LIN {X -0.079,Y -462.079,Z 459.993,A 0.000,B 0.000,C 90.000,E1 214.659} C_DIS
LIN {X 0.017,Y -457.566,Z 459.980,A 0.000,B 0.000,C 90.000,E1 212.418} C_DIS
LIN {X -0.236,Y -453.208,Z 459.968,A 0.000,B 0.000,C 90.000,E1 210.207} C_DIS
LIN {X 0.089,Y -449.505,Z 459.957,A 0.000,B 0.000,C 90.000,E1 208.231} C_DIS
LIN {X 0.041,Y -446.412,Z 459.948,A 0.000,B 0.000,C 90.000,E1 206.616} C_DIS
LIN {X 0.179,Y -442.573,Z 459.937,A 0.000,B 0.000,C 90.000,E1 204.643} C_DIS
LIN {X -0.081,Y -440.644,Z 459.932,A 0.000,B 0.000,C 90.000,E1 203.695} C_DIS
LIN {X -0.199,Y -436.151,Z 459.919,A 0.000,B 0.000,C 90.000,E1 201.408} C_DIS
LIN {X -0.233,Y -433.117,Z 459.910,A 0.000,B 0.000,C 90.000,E1 199.758} C_DIS
LIN {X -0.033,Y -429.082,Z 459.897,A 0.000,B 0.000,C 90.000,E1 197.402} C_DIS
LIN {X 0.001,Y -424.902,Z 459.882,A 0.000,B 0.000,C 90.000,E1 194.717} C_DIS
LIN {X -0.050,Y -422.064,Z 459.871,A 0.000,B 0.000,C 90.000,E1 192.703} C_DIS
LIN {X -0.165,Y -418.201,Z 459.854,A 0.000,B 0.000,C 90.000,E1 189.670} C_DIS
LIN {X 0.173,Y -415.396,Z 459.840,A 0.000,B 0.000,C 90.000,E1 187.239} C_DIS
LIN {X -0.106,Y -413.960,Z 459.833,A 0.000,B 0.000,C 90.000,E1 185.910} C_DIS
LIN {X -0.021,Y -411.212,Z 459.818,A 0.000,B 0.000,C 90.000,E1 183.154} C_DIS
LIN {X -0.018,Y -409.551,Z 459.806,A 0.000,B 0.000,C 90.000,E1 181.088} C_DIS
LIN {X -0.128,Y -407.489,Z 459.787,A 0.000,B 0.000,C 90.000,E1 177.650} C_DIS
LIN {X 0.157,Y -406.307,Z 459.766,A 0.000,B 0.000,C 90.000,E1 173.799} C_DIS
LIN {X 0.171,Y -406.510,Z 459.745,A 0.000,B 0.000,C 90.000,E1 169.982} C_DIS
LIN {X 0.162,Y -407.845,Z 459.723,A 0.000,B 0.000,C 90.000,E1 166.172} C_DIS
LIN {X 0.133,Y -408.980,Z 459.712,A 0.000,B 0.000,C 90.000,E1 164.102} C_DIS
LIN {X 0.093,Y -411.915,Z 459.691,A 0.000,B 0.000,C 90.000,E1 160.315} C_DIS
LIN {X -0.064,Y -414.691,Z 459.676,A 0.000,B 0.000,C 90.000,E1 157.592} C_DIS
LIN {X 0.044,Y -417.933,Z 459.660,A 0.000,B 0.000,C 90.000,E1 154.845} C_DIS
LIN {X 0.167,Y -420.127,Z 459.651,A 0.000,B 0.000,C 90.000,E1 153.127} C_DIS
LIN {X -0.114,Y -423.324,Z 459.638,A 0.000,B 0.000,C 90.000,E1 150.795} C_DIS
LIN {X 0.121,Y -426.091,Z 459.626,A 0.000,B 0.000,C 90.000,E1 148.742} C_DIS
LIN {X -0.070,Y -428.532,Z 459.617,A 0.000,B 0.000,C 90.000,E1 147.089} C_DIS
LIN {X 0.148,Y -431.633,Z 459.606,A 0.000,B 0.000,C 90.000,E1 145.055} C_DIS
LIN {X -0.120,Y -435.369,Z 459.593,A 0.000,B 0.000,C 90.000,E1 142.763} C_DIS
LIN {X -0.066,Y -439.785,Z 459.578,A 0.000,B 0.000,C 90.000,E1 140.114} C_DIS
LIN {X -0.206,Y -443.193,Z 459.567,A 0.000,B 0.000,C 90.000,E1 138.162} C_DIS
LIN {X 0.028,Y -445.355,Z 459.560,A 0.000,B 0.000,C 90.000,E1 136.824} C_DIS
LIN {X -0.015,Y -447.307,Z 459.553,A 0.000,B 0.000,C 90.000,E1 135.526} C_DIS
LIN {X -0.039,Y -448.476,Z 459.548,A 0.000,B 0.000,C 90.000,E1 134.555} C_DIS
LIN {X 0.276,Y -449.230,Z 459.544,A 0.000,B 0.000,C 90.000,E1 133.866} C_DIS
LIN {X -0.030,Y -450.411,Z 459.537,A 0.000,B 0.000,C 90.000,E1 132.609} C_DIS
LIN {X 0.014,Y -451.134,Z 459.530,A 0.000,B 0.000,C 90.000,E1 131.310} C_DIS
LIN {X 0.068,Y -451.303,Z 459.524,A 0.000,B 0.000,C 90.000,E1 130.334} C_DIS
LIN {X -0.221,Y -451.124,Z 459.521,A 0.000,B 0.000,C 90.000,E1 129.725} C_DIS
LIN {X 0.119,Y -450.766,Z 459.517,A 0.000,B 0.000,C 90.000,E1 129.036} C_DIS
LIN {X 0.172,Y -450.342,Z 459.513,A 0.000,B 0.000,C 90.000,E1 128.382} C_DIS
LIN {X -0.003,Y -448.898,Z 459.506,A 0.000,B 0.000,C 90.000,E1 127.111} C_DIS
LIN {X 0.008,Y -447.522,Z 459.501,A 0.000,B 0.000,C 90.000,E1 126.137} C_DIS
LIN {X -0.229,Y -446.452,Z 459.497,A 0.000,B 0.000,C 90.000,E1 125.518} C_DIS
LIN {X -0.154,Y -444.523,Z 459.492,A 0.000,B 0.000,C 90.000,E1 124.532} C_DIS
LIN {X -0.057,Y -441.550,Z 459.485,A 0.000,B 0.000,C 90.000,E1 123.214} C_DIS
LIN {X 0.124,Y -438.283,Z 459.477,A 0.000,B 0.000,C 90.000,E1 121.878} C_DIS
LIN {X -0.117,Y -434.841,Z 459.470,A 0.000,B 0.000,C 90.000,E1 120.590} C_DIS
LIN {X 0.122,Y -432.255,Z 459.465,A 0.000,B 0.000,C 90.000,E1 119.617} C_DIS
LIN {X 0.083,Y -432.255,Z 459.465,A 0.000,B 0.000,C 90.000,E1 119.617} C_DIS
LIN {X 0.136,Y -441.772,Z 459.444,A 0.000,B 0.000,C 90.000,E1 115.924} C_DIS
LIN {X 0.059,Y -444.699,Z 459.439,A 0.000,B 0.000,C 90.000,E1 114.951} C_DIS
LIN {X 0.031,Y -454.671,Z 459.415,A 0.000,B 0.000,C 90.000,E1 110.737} C_DIS
LIN {X 0.153,Y -457.324,Z 459.410,A 0.000,B 0.000,C 90.000,E1 109.758} C_DIS
LIN {X -0.209,Y -465.949,Z 459.387,A 0.000,B 0.000,C 90.000,E1 105.662} C_DIS
LIN {X -0.038,Y -467.513,Z 459.383,A 0.000,B 0.000,C 90.000,E1 105.009} C_DIS
LIN {X -0.234,Y -468.096,Z 459.382,A 0.000,B 0.000,C 90.000,E1 104.717} C_DIS
LIN {X -0.094,Y -475.756,Z 459.357,A 0.000,B 0.000,C 90.000,E1 100.310} C_DIS
LIN {X 0.211,Y -476.285,Z 459.356,A 0.000,B 0.000,C 90.000,E1 99.962} C_DIS
LIN {X 0.208,Y -479.372,Z 459.340,A 0.000,B 0.000,C 90.000,E1 97.239} C_DIS
LIN {X 0.188,Y -558.722,Z 459.340,A 0.000,B 0.000,C 90.000,E1 97.239} C_DIS
LIN {X 0.091,Y -564.116,Z 459.340,A 0.000,B 0.000,C 90.000,E1 97.182} C_DIS
LIN {X 0.113,Y -570.120,Z 459.339,A 0.000,B 0.000,C 90.000,E1 97.068} C_DIS
LIN {X -0.229,Y -576.419,Z 459.339,A 0.000,B 0.000,C 90.000,E1 96.947} C_DIS
LIN {X 0.097,Y -582.845,Z 459.337,A 0.000,B 0.000,C 90.000,E1 96.720} C_DIS
LIN {X 0.040,Y -589.213,Z 459.336,A 0.000,B 0.000,C 90.000,E1 96.486} C_DIS
LIN {X 0.176,Y -595.796,Z 459.335,A 0.000,B 0.000,C 90.000,E1 96.201} C_DIS
LIN {X -0.029,Y -601.591,Z 459.333,A 0.000,B 0.000,C 90.000,E1 95.910} C_DIS
LIN {X -0.209,Y -607.593,Z 459.331,A 0.000,B 0.000,C 90.000,E1 95.568} C_DIS
LIN {X -0.076,Y -613.091,Z 459.329,A 0.000,B 0.000,C 90.000,E1 95.163} C_DIS
LIN {X 0.014,Y -614.544,Z 459.328,A 0.000,B 0.000,C 90.000,E1 95.049} C_DIS
LIN {X -0.034,Y -620.912,Z 459.325,A 0.000,B 0.000,C 90.000,E1 94.473} C_DIS
LIN {X 0.204,Y -625.161,Z 459.322,A 0.000,B 0.000,C 90.000,E1 93.955} C_DIS
LIN {X -0.090,Y -627.282,Z 459.321,A 0.000,B 0.000,C 90.000,E1 93.726} C_DIS
LIN {X 0.250,Y -628.777,Z 459.319,A 0.000,B 0.000,C 90.000,E1 93.440} C_DIS
LIN {X -0.269,Y -631.451,Z 459.316,A 0.000,B 0.000,C 90.000,E1 92.980} C_DIS
LIN {X -0.179,Y -633.775,Z 459.314,A 0.000,B 0.000,C 90.000,E1 92.465} C_DIS
LIN {X -0.306,Y -635.760,Z 459.309,A 0.000,B 0.000,C 90.000,E1 91.718} C_DIS
LIN {X -0.181,Y -636.632,Z 459.307,A 0.000,B 0.000,C 90.000,E1 91.203} C_DIS
LIN {X -0.048,Y -637.073,Z 459.304,A 0.000,B 0.000,C 90.000,E1 90.688} C_DIS
LIN {X 0.091,Y -637.071,Z 459.301,A 0.000,B 0.000,C 90.000,E1 90.172} C_DIS
LIN {X -0.158,Y -636.918,Z 459.300,A 0.000,B 0.000,C 90.000,E1 89.943} C_DIS
LIN {X -0.019,Y -636.261,Z 459.297,A 0.000,B 0.000,C 90.000,E1 89.427} C_DIS
LIN {X 0.114,Y -635.024,Z 459.294,A 0.000,B 0.000,C 90.000,E1 88.912} C_DIS
LIN {X 0.238,Y -633.501,Z 459.291,A 0.000,B 0.000,C 90.000,E1 88.396} C_DIS
LIN {X -0.001,Y -632.517,Z 459.290,A 0.000,B 0.000,C 90.000,E1 88.165} C_DIS
LIN {X 0.107,Y -629.929,Z 459.287,A 0.000,B 0.000,C 90.000,E1 87.650} C_DIS
LIN {X 0.050,Y -626.107,Z 459.284,A 0.000,B 0.000,C 90.000,E1 87.020} C_DIS
LIN {X -0.153,Y -620.658,Z 459.279,A 0.000,B 0.000,C 90.000,E1 86.274} C_DIS
LIN {X -0.250,Y -615.157,Z 459.276,A 0.000,B 0.000,C 90.000,E1 85.641} C_DIS
LIN {X -0.065,Y -609.946,Z 459.273,A 0.000,B 0.000,C 90.000,E1 85.122} C_DIS
LIN {X -0.133,Y -608.649,Z 459.272,A 0.000,B 0.000,C 90.000,E1 85.008} C_DIS
LIN {X -0.109,Y -603.026,Z 459.270,A 0.000,B 0.000,C 90.000,E1 84.546} C_DIS
LIN {X 0.081,Y -598.091,Z 459.268,A 0.000,B 0.000,C 90.000,E1 84.204} C_DIS
LIN {X -0.141,Y -594.766,Z 459.267,A 0.000,B 0.000,C 90.000,E1 84.033} C_DIS
LIN {X -0.035,Y -588.527,Z 459.265,A 0.000,B 0.000,C 90.000,E1 83.685} C_DIS
LIN {X -0.071,Y -585.000,Z 459.264,A 0.000,B 0.000,C 90.000,E1 83.514} C_DIS
LIN {X -0.245,Y -583.090,Z 459.264,A 0.000,B 0.000,C 90.000,E1 83.451} C_DIS
LIN {X 0.093,Y -577.795,Z 459.262,A 0.000,B 0.000,C 90.000,E1 83.223} C_DIS
LIN {X -0.016,Y -571.567,Z 459.261,A 0.000,B 0.000,C 90.000,E1 83.053} C_DIS
LIN {X 0.061,Y -564.953,Z 459.261,A 0.000,B 0.000,C 90.000,E1 82.932} C_DIS
LIN {X 0.160,Y -559.170,Z 459.261,A 0.000,B 0.000,C 90.000,E1 82.875} C_DIS
LIN {X 0.104,Y -484.840,Z 459.261,A 0.000,B 0.000,C 90.000,E1 82.875} C_DIS
LIN {X -0.113,Y -484.690,Z 459.254,A 0.000,B 0.000,C 90.000,E1 81.659} C_DIS
LIN {X -0.099,Y -483.703,Z 459.249,A 0.000,B 0.000,C 90.000,E1 80.735} C_DIS
LIN {X 0.265,Y -480.630,Z 459.228,A 0.000,B 0.000,C 90.000,E1 76.992} C_DIS
LIN {X 0.123,Y -480.315,Z 459.226,A 0.000,B 0.000,C 90.000,E1 76.700} C_DIS
LIN {X 0.026,Y -474.131,Z 459.200,A 0.000,B 0.000,C 90.000,E1 72.054} C_DIS
LIN {X -0.105,Y -465.601,Z 459.172,A 0.000,B 0.000,C 90.000,E1 67.050} C_DIS
LIN {X -0.108,Y -458.658,Z 459.154,A 0.000,B 0.000,C 90.000,E1 63.768} C_DIS
LIN {X -0.147,Y -458.658,Z 459.154,A 0.000,B 0.000,C 90.000,E1 63.768} C_DIS
LIN {X -0.198,Y -466.432,Z 459.148,A 0.000,B 0.000,C 90.000,E1 62.615} C_DIS
LIN {X -0.201,Y -473.768,Z 459.142,A 0.000,B 0.000,C 90.000,E1 61.513} C_DIS
LIN {X 0.126,Y -480.526,Z 459.136,A 0.000,B 0.000,C 90.000,E1 60.383} C_DIS
LIN {X 0.085,Y -484.924,Z 459.131,A 0.000,B 0.000,C 90.000,E1 59.616} C_DIS
LIN {X 0.123,Y -488.077,Z 459.128,A 0.000,B 0.000,C 90.000,E1 58.997} C_DIS
LIN {X -0.021,Y -491.497,Z 459.124,A 0.000,B 0.000,C 90.000,E1 58.250} C_DIS
LIN {X -0.189,Y -493.935,Z 459.120,A 0.000,B 0.000,C 90.000,E1 57.661} C_DIS
LIN {X -0.077,Y -495.986,Z 459.117,A 0.000,B 0.000,C 90.000,E1 57.041} C_DIS
LIN {X -0.087,Y -498.471,Z 459.112,A 0.000,B 0.000,C 90.000,E1 56.135} C_DIS
LIN {X 0.063,Y -499.755,Z 459.109,A 0.000,B 0.000,C 90.000,E1 55.515} C_DIS
LIN {X 0.098,Y -501.142,Z 459.103,A 0.000,B 0.000,C 90.000,E1 54.609} C_DIS
LIN {X 0.147,Y -502.283,Z 459.098,A 0.000,B 0.000,C 90.000,E1 53.703} C_DIS
LIN {X -0.200,Y -502.907,Z 459.094,A 0.000,B 0.000,C 90.000,E1 52.844} C_DIS
LIN {X 0.053,Y -503.314,Z 459.087,A 0.000,B 0.000,C 90.000,E1 51.618} C_DIS
LIN {X 0.029,Y -503.403,Z 459.082,A 0.000,B 0.000,C 90.000,E1 50.723} C_DIS
LIN {X 0.124,Y -503.387,Z 459.079,A 0.000,B 0.000,C 90.000,E1 50.114} C_DIS
LIN {X 0.104,Y -503.125,Z 459.074,A 0.000,B 0.000,C 90.000,E1 49.218} C_DIS
LIN {X -0.331,Y -502.312,Z 459.064,A 0.000,B 0.000,C 90.000,E1 47.472} C_DIS
LIN {X 0.177,Y -501.600,Z 459.057,A 0.000,B 0.000,C 90.000,E1 46.215} C_DIS
LIN {X -0.185,Y -500.627,Z 459.049,A 0.000,B 0.000,C 90.000,E1 44.757} C_DIS
LIN {X -0.065,Y -499.708,Z 459.042,A 0.000,B 0.000,C 90.000,E1 43.542} C_DIS
LIN {X -0.108,Y -498.547,Z 459.034,A 0.000,B 0.000,C 90.000,E1 42.043} C_DIS
LIN {X 0.050,Y -497.041,Z 459.023,A 0.000,B 0.000,C 90.000,E1 40.216} C_DIS
LIN {X 0.236,Y -495.466,Z 459.013,A 0.000,B 0.000,C 90.000,E1 38.382} C_DIS
LIN {X 0.086,Y -493.825,Z 459.003,A 0.000,B 0.000,C 90.000,E1 36.583} C_DIS
LIN {X -0.094,Y -492.591,Z 458.997,A 0.000,B 0.000,C 90.000,E1 35.391} C_DIS
LIN {X -0.038,Y -490.933,Z 458.988,A 0.000,B 0.000,C 90.000,E1 33.865} C_DIS
LIN {X -0.018,Y -489.233,Z 458.980,A 0.000,B 0.000,C 90.000,E1 32.339} C_DIS
LIN {X 0.114,Y -487.317,Z 458.971,A 0.000,B 0.000,C 90.000,E1 30.797} C_DIS
LIN {X -0.028,Y -485.783,Z 458.964,A 0.000,B 0.000,C 90.000,E1 29.589} C_DIS
LIN {X -0.221,Y -483.471,Z 458.954,A 0.000,B 0.000,C 90.000,E1 27.769} C_DIS
LIN {X -0.054,Y -480.630,Z 458.940,A 0.000,B 0.000,C 90.000,E1 25.283} C_DIS
LIN {X -0.176,Y -478.269,Z 458.927,A 0.000,B 0.000,C 90.000,E1 22.823} C_DIS
LIN {X 0.159,Y -476.710,Z 458.915,A 0.000,B 0.000,C 90.000,E1 20.610} C_DIS
LIN {X -0.137,Y -475.497,Z 458.904,A 0.000,B 0.000,C 90.000,E1 18.779} C_DIS
LIN {X -0.130,Y -474.555,Z 458.896,A 0.000,B 0.000,C 90.000,E1 17.221} C_DIS
LIN {X 0.096,Y -473.109,Z 458.883,A 0.000,B 0.000,C 90.000,E1 15.009} C_DIS
LIN {X -0.097,Y -471.382,Z 458.864,A 0.000,B 0.000,C 90.000,E1 11.591} C_DIS
LIN {X 0.198,Y -470.425,Z 458.845,A 0.000,B 0.000,C 90.000,E1 8.106} C_DIS
LIN {X -0.196,Y -470.501,Z 458.826,A 0.000,B 0.000,C 90.000,E1 4.702} C_DIS
LIN {X -0.231,Y -472.150,Z 458.803,A 0.000,B 0.000,C 90.000,E1 0.630} C_DIS
LIN {X 0.218,Y -473.164,Z 458.795,A 0.000,B 0.000,C 90.000,E1 359.141} C_DIS
LIN {X 0.223,Y -475.718,Z 458.780,A 0.000,B 0.000,C 90.000,E1 356.331} C_DIS
LIN {X -0.096,Y -479.014,Z 458.764,A 0.000,B 0.000,C 90.000,E1 353.571} C_DIS
LIN {X 0.150,Y -481.944,Z 458.752,A 0.000,B 0.000,C 90.000,E1 351.376} C_DIS
LIN {X 0.158,Y -485.257,Z 458.740,A 0.000,B 0.000,C 90.000,E1 349.218} C_DIS
LIN {X -0.088,Y -491.443,Z 458.722,A 0.000,B 0.000,C 90.000,E1 345.880} C_DIS
LIN {X 0.038,Y -496.067,Z 458.710,A 0.000,B 0.000,C 90.000,E1 343.740} C_DIS
LIN {X -0.044,Y -501.143,Z 458.698,A 0.000,B 0.000,C 90.000,E1 341.638} C_DIS
LIN {X 0.165,Y -506.451,Z 458.686,A 0.000,B 0.000,C 90.000,E1 339.518} C_DIS
LIN {X 0.096,Y -511.096,Z 458.676,A 0.000,B 0.000,C 90.000,E1 337.741} C_DIS
LIN {X 0.053,Y -515.667,Z 458.667,A 0.000,B 0.000,C 90.000,E1 335.973} C_DIS
LIN {X -0.235,Y -519.412,Z 458.658,A 0.000,B 0.000,C 90.000,E1 334.537} C_DIS
LIN {X 0.140,Y -523.946,Z 458.649,A 0.000,B 0.000,C 90.000,E1 332.743} C_DIS
LIN {X -0.209,Y -529.892,Z 458.636,A 0.000,B 0.000,C 90.000,E1 330.461} C_DIS
LIN {X 0.159,Y -535.227,Z 458.625,A 0.000,B 0.000,C 90.000,E1 328.408} C_DIS
LIN {X 0.023,Y -539.779,Z 458.615,A 0.000,B 0.000,C 90.000,E1 326.707} C_DIS
LIN {X -0.188,Y -543.602,Z 458.607,A 0.000,B 0.000,C 90.000,E1 325.308} C_DIS
LIN {X -0.240,Y -549.057,Z 458.596,A 0.000,B 0.000,C 90.000,E1 323.336} C_DIS
LIN {X 0.102,Y -553.814,Z 458.587,A 0.000,B 0.000,C 90.000,E1 321.618} C_DIS
LIN {X 0.196,Y -560.142,Z 458.574,A 0.000,B 0.000,C 90.000,E1 319.380} C_DIS
LIN {X -0.157,Y -564.970,Z 458.565,A 0.000,B 0.000,C 90.000,E1 317.757} C_DIS
LIN {X -0.106,Y -568.885,Z 458.558,A 0.000,B 0.000,C 90.000,E1 316.377} C_DIS
LIN {X 0.215,Y -574.285,Z 458.547,A 0.000,B 0.000,C 90.000,E1 314.433} C_DIS
LIN {X -0.267,Y -578.948,Z 458.538,A 0.000,B 0.000,C 90.000,E1 312.852} C_DIS
LIN {X 0.039,Y -582.833,Z 458.530,A 0.000,B 0.000,C 90.000,E1 311.472} C_DIS
LIN {X -0.033,Y -586.689,Z 458.523,A 0.000,B 0.000,C 90.000,E1 310.135} C_DIS
LIN {X -0.095,Y -589.734,Z 458.517,A 0.000,B 0.000,C 90.000,E1 309.072} C_DIS
LIN {X 0.016,Y -593.385,Z 458.510,A 0.000,B 0.000,C 90.000,E1 307.729} C_DIS
LIN {X 0.066,Y -596.294,Z 458.504,A 0.000,B 0.000,C 90.000,E1 306.664} C_DIS
LIN {X -0.092,Y -599.857,Z 458.496,A 0.000,B 0.000,C 90.000,E1 305.358} C_DIS
LIN {X 0.194,Y -602.579,Z 458.491,A 0.000,B 0.000,C 90.000,E1 304.278} C_DIS
LIN {X 0.031,Y -605.197,Z 458.485,A 0.000,B 0.000,C 90.000,E1 303.245} C_DIS
LIN {X -0.100,Y -607.702,Z 458.479,A 0.000,B 0.000,C 90.000,E1 302.212} C_DIS
LIN {X -0.307,Y -611.284,Z 458.470,A 0.000,B 0.000,C 90.000,E1 300.669} C_DIS
LIN {X 0.114,Y -614.013,Z 458.463,A 0.000,B 0.000,C 90.000,E1 299.333} C_DIS
LIN {X 0.277,Y -616.687,Z 458.456,A 0.000,B 0.000,C 90.000,E1 298.025} C_DIS
LIN {X 0.189,Y -619.833,Z 458.447,A 0.000,B 0.000,C 90.000,E1 296.488} C_DIS
LIN {X 0.171,Y -621.298,Z 458.443,A 0.000,B 0.000,C 90.000,E1 295.720} C_DIS
LIN {X -0.093,Y -623.968,Z 458.434,A 0.000,B 0.000,C 90.000,E1 294.207} C_DIS
LIN {X 0.258,Y -625.952,Z 458.427,A 0.000,B 0.000,C 90.000,E1 292.898} C_DIS
LIN {X -0.166,Y -628.104,Z 458.419,A 0.000,B 0.000,C 90.000,E1 291.408} C_DIS
LIN {X 0.018,Y -629.794,Z 458.412,A 0.000,B 0.000,C 90.000,E1 290.120} C_DIS
LIN {X 0.019,Y -631.360,Z 458.405,A 0.000,B 0.000,C 90.000,E1 288.852} C_DIS
LIN {X 0.050,Y -632.768,Z 458.398,A 0.000,B 0.000,C 90.000,E1 287.583} C_DIS
LIN {X -0.088,Y -634.202,Z 458.389,A 0.000,B 0.000,C 90.000,E1 286.079} C_DIS
LIN {X -0.017,Y -634.817,Z 458.385,A 0.000,B 0.000,C 90.000,E1 285.315} C_DIS
LIN {X -0.297,Y -635.887,Z 458.377,A 0.000,B 0.000,C 90.000,E1 283.828} C_DIS
LIN {X 0.074,Y -636.469,Z 458.370,A 0.000,B 0.000,C 90.000,E1 282.535} C_DIS
LIN {X 0.002,Y -636.857,Z 458.364,A 0.000,B 0.000,C 90.000,E1 281.535} C_DIS
LIN {X 0.257,Y -637.126,Z 458.357,A 0.000,B 0.000,C 90.000,E1 280.254} C_DIS
LIN {X -0.112,Y -637.081,Z 458.350,A 0.000,B 0.000,C 90.000,E1 279.029} C_DIS
LIN {X 0.229,Y -636.921,Z 458.345,A 0.000,B 0.000,C 90.000,E1 277.992} C_DIS
LIN {X 0.023,Y -636.491,Z 458.339,A 0.000,B 0.000,C 90.000,E1 277.004} C_DIS
LIN {X -0.074,Y -636.007,Z 458.335,A 0.000,B 0.000,C 90.000,E1 276.258} C_DIS
LIN {X 0.258,Y -635.175,Z 458.329,A 0.000,B 0.000,C 90.000,E1 275.220} C_DIS
LIN {X 0.153,Y -634.309,Z 458.325,A 0.000,B 0.000,C 90.000,E1 274.473} C_DIS
LIN {X -0.223,Y -632.945,Z 458.319,A 0.000,B 0.000,C 90.000,E1 273.498} C_DIS
LIN {X -0.250,Y -630.965,Z 458.312,A 0.000,B 0.000,C 90.000,E1 272.236} C_DIS
LIN {X 0.314,Y -628.647,Z 458.305,A 0.000,B 0.000,C 90.000,E1 270.917} C_DIS
LIN {X 0.194,Y -626.139,Z 458.298,A 0.000,B 0.000,C 90.000,E1 269.656} C_DIS
LIN {X 0.030,Y -623.442,Z 458.291,A 0.000,B 0.000,C 90.000,E1 268.396} C_DIS
LIN {X -0.165,Y -620.490,Z 458.284,A 0.000,B 0.000,C 90.000,E1 267.135} C_DIS
LIN {X 0.249,Y -617.421,Z 458.277,A 0.000,B 0.000,C 90.000,E1 265.812} C_DIS
LIN {X -0.026,Y -615.558,Z 458.273,A 0.000,B 0.000,C 90.000,E1 265.065} C_DIS
LIN {X 0.307,Y -612.250,Z 458.265,A 0.000,B 0.000,C 90.000,E1 263.742} C_DIS
LIN {X -0.295,Y -609.623,Z 458.260,A 0.000,B 0.000,C 90.000,E1 262.761} C_DIS
LIN {X -0.001,Y -606.148,Z 458.252,A 0.000,B 0.000,C 90.000,E1 261.432} C_DIS
LIN {X -0.275,Y -602.664,Z 458.245,A 0.000,B 0.000,C 90.000,E1 260.151} C_DIS
LIN {X 0.273,Y -599.738,Z 458.239,A 0.000,B 0.000,C 90.000,E1 259.050} C_DIS
LIN {X 0.006,Y -594.420,Z 458.229,A 0.000,B 0.000,C 90.000,E1 257.229} C_DIS
LIN {X 0.233,Y -590.449,Z 458.222,A 0.000,B 0.000,C 90.000,E1 255.880} C_DIS
LIN {X 0.276,Y -587.280,Z 458.216,A 0.000,B 0.000,C 90.000,E1 254.810} C_DIS
LIN {X 0.278,Y -584.000,Z 458.210,A 0.000,B 0.000,C 90.000,E1 253.740} C_DIS
LIN {X 0.228,Y -580.693,Z 458.204,A 0.000,B 0.000,C 90.000,E1 252.670} C_DIS
LIN {X -0.244,Y -577.325,Z 458.198,A 0.000,B 0.000,C 90.000,E1 251.638} C_DIS
LIN {X -0.210,Y -573.874,Z 458.192,A 0.000,B 0.000,C 90.000,E1 250.550} C_DIS
LIN {X -0.031,Y -570.334,Z 458.186,A 0.000,B 0.000,C 90.000,E1 249.444} C_DIS
LIN {X -0.295,Y -565.802,Z 458.178,A 0.000,B 0.000,C 90.000,E1 248.103} C_DIS
LIN {X -0.016,Y -561.956,Z 458.172,A 0.000,B 0.000,C 90.000,E1 246.975} C_DIS
LIN {X -0.225,Y -556.948,Z 458.164,A 0.000,B 0.000,C 90.000,E1 245.613} C_DIS
LIN {X 0.159,Y -552.860,Z 458.158,A 0.000,B 0.000,C 90.000,E1 244.460} C_DIS
LIN {X 0.006,Y -547.692,Z 458.150,A 0.000,B 0.000,C 90.000,E1 243.076} C_DIS
LIN {X -0.004,Y -540.403,Z 458.139,A 0.000,B 0.000,C 90.000,E1 241.101} C_DIS
LIN {X 0.117,Y -535.302,Z 458.132,A 0.000,B 0.000,C 90.000,E1 239.665} C_DIS
LIN {X 0.100,Y -529.219,Z 458.122,A 0.000,B 0.000,C 90.000,E1 237.946} C_DIS
LIN {X 0.065,Y -523.158,Z 458.112,A 0.000,B 0.000,C 90.000,E1 236.215} C_DIS
LIN {X -0.037,Y -518.073,Z 458.104,A 0.000,B 0.000,C 90.000,E1 234.769} C_DIS
LIN {X -0.015,Y -511.827,Z 458.095,A 0.000,B 0.000,C 90.000,E1 233.004} C_DIS
LIN {X -0.243,Y -500.491,Z 458.075,A 0.000,B 0.000,C 90.000,E1 229.461} C_DIS
LIN {X -0.057,Y -495.153,Z 458.065,A 0.000,B 0.000,C 90.000,E1 227.634} C_DIS
LIN {X 0.145,Y -489.132,Z 458.053,A 0.000,B 0.000,C 90.000,E1 225.486} C_DIS
LIN {X -0.159,Y -483.326,Z 458.041,A 0.000,B 0.000,C 90.000,E1 223.380} C_DIS
LIN {X -0.037,Y -478.500,Z 458.031,A 0.000,B 0.000,C 90.000,E1 221.515} C_DIS
LIN {X -0.106,Y -472.498,Z 458.017,A 0.000,B 0.000,C 90.000,E1 219.036} C_DIS
LIN {X 0.081,Y -466.776,Z 458.003,A 0.000,B 0.000,C 90.000,E1 216.503} C_DIS
LIN {X -0.088,Y -463.431,Z 457.994,A 0.000,B 0.000,C 90.000,E1 214.945} C_DIS
LIN {X -0.218,Y -458.209,Z 457.980,A 0.000,B 0.000,C 90.000,E1 212.418} C_DIS
LIN {X 0.167,Y -453.831,Z 457.968,A 0.000,B 0.000,C 90.000,E1 210.129} C_DIS
LIN {X -0.112,Y -450.078,Z 457.957,A 0.000,B 0.000,C 90.000,E1 208.231} C_DIS
LIN {X -0.147,Y -446.989,Z 457.948,A 0.000,B 0.000,C 90.000,E1 206.616} C_DIS
LIN {X -0.136,Y -442.490,Z 457.935,A 0.000,B 0.000,C 90.000,E1 204.335} C_DIS
LIN {X -0.030,Y -437.922,Z 457.922,A 0.000,B 0.000,C 90.000,E1 202.025} C_DIS
LIN {X -0.201,Y -434.232,Z 457.911,A 0.000,B 0.000,C 90.000,E1 200.066} C_DIS
LIN {X 0.165,Y -430.094,Z 457.898,A 0.000,B 0.000,C 90.000,E1 197.692} C_DIS
LIN {X 0.219,Y -425.850,Z 457.884,A 0.000,B 0.000,C 90.000,E1 195.009} C_DIS
LIN {X 0.091,Y -422.938,Z 457.872,A 0.000,B 0.000,C 90.000,E1 193.008} C_DIS
LIN {X 0.097,Y -418.963,Z 457.855,A 0.000,B 0.000,C 90.000,E1 189.962} C_DIS
LIN {X -0.008,Y -416.504,Z 457.844,A 0.000,B 0.000,C 90.000,E1 187.936} C_DIS
LIN {X -0.174,Y -414.304,Z 457.833,A 0.000,B 0.000,C 90.000,E1 185.910} C_DIS
LIN {X -0.077,Y -411.557,Z 457.818,A 0.000,B 0.000,C 90.000,E1 183.154} C_DIS
LIN {X -0.066,Y -409.863,Z 457.806,A 0.000,B 0.000,C 90.000,E1 181.088} C_DIS
LIN {X -0.163,Y -407.814,Z 457.787,A 0.000,B 0.000,C 90.000,E1 177.650} C_DIS
LIN {X 0.101,Y -406.617,Z 457.764,A 0.000,B 0.000,C 90.000,E1 173.457} C_DIS
LIN {X 0.167,Y -406.864,Z 457.745,A 0.000,B 0.000,C 90.000,E1 169.982} C_DIS
LIN {X 0.174,Y -408.233,Z 457.723,A 0.000,B 0.000,C 90.000,E1 166.172} C_DIS
LIN {X 0.155,Y -409.379,Z 457.712,A 0.000,B 0.000,C 90.000,E1 164.102} C_DIS
LIN {X 0.133,Y -412.347,Z 457.691,A 0.000,B 0.000,C 90.000,E1 160.315} C_DIS
LIN {X 0.078,Y -414.761,Z 457.677,A 0.000,B 0.000,C 90.000,E1 157.922} C_DIS
LIN {X 0.032,Y -417.575,Z 457.664,A 0.000,B 0.000,C 90.000,E1 155.537} C_DIS
LIN {X -0.128,Y -420.664,Z 457.651,A 0.000,B 0.000,C 90.000,E1 153.179} C_DIS
LIN {X -0.041,Y -424.416,Z 457.636,A 0.000,B 0.000,C 90.000,E1 150.461} C_DIS
LIN {X -0.153,Y -427.750,Z 457.623,A 0.000,B 0.000,C 90.000,E1 148.122} C_DIS
LIN {X 0.047,Y -431.338,Z 457.610,A 0.000,B 0.000,C 90.000,E1 145.754} C_DIS
LIN {X 0.198,Y -433.507,Z 457.602,A 0.000,B 0.000,C 90.000,E1 144.402} C_DIS
LIN {X 0.059,Y -436.825,Z 457.591,A 0.000,B 0.000,C 90.000,E1 142.431} C_DIS
LIN {X 0.181,Y -440.195,Z 457.580,A 0.000,B 0.000,C 90.000,E1 140.436} C_DIS
LIN {X 0.106,Y -441.952,Z 457.575,A 0.000,B 0.000,C 90.000,E1 139.461} C_DIS
LIN {X -0.002,Y -444.871,Z 457.566,A 0.000,B 0.000,C 90.000,E1 137.838} C_DIS
LIN {X -0.030,Y -446.601,Z 457.560,A 0.000,B 0.000,C 90.000,E1 136.863} C_DIS
LIN {X -0.067,Y -448.602,Z 457.553,A 0.000,B 0.000,C 90.000,E1 135.567} C_DIS
LIN {X -0.071,Y -449.479,Z 457.550,A 0.000,B 0.000,C 90.000,E1 134.919} C_DIS
LIN {X -0.064,Y -450.668,Z 457.544,A 0.000,B 0.000,C 90.000,E1 133.947} C_DIS
LIN {X 0.288,Y -451.958,Z 457.537,A 0.000,B 0.000,C 90.000,E1 132.609} C_DIS
LIN {X 0.019,Y -452.794,Z 457.530,A 0.000,B 0.000,C 90.000,E1 131.353} C_DIS
LIN {X 0.086,Y -452.998,Z 457.524,A 0.000,B 0.000,C 90.000,E1 130.378} C_DIS
LIN {X -0.130,Y -452.771,Z 457.519,A 0.000,B 0.000,C 90.000,E1 129.439} C_DIS
LIN {X 0.225,Y -452.366,Z 457.515,A 0.000,B 0.000,C 90.000,E1 128.749} C_DIS
LIN {X 0.291,Y -451.846,Z 457.512,A 0.000,B 0.000,C 90.000,E1 128.096} C_DIS
LIN {X 0.067,Y -450.752,Z 457.507,A 0.000,B 0.000,C 90.000,E1 127.156} C_DIS
LIN {X -0.170,Y -449.390,Z 457.501,A 0.000,B 0.000,C 90.000,E1 126.217} C_DIS
LIN {X 0.235,Y -448.380,Z 457.498,A 0.000,B 0.000,C 90.000,E1 125.518} C_DIS
LIN {X 0.076,Y -446.440,Z 457.492,A 0.000,B 0.000,C 90.000,E1 124.565} C_DIS
LIN {X 0.089,Y -445.031,Z 457.489,A 0.000,B 0.000,C 90.000,E1 123.913} C_DIS
LIN {X -0.047,Y -441.826,Z 457.481,A 0.000,B 0.000,C 90.000,E1 122.625} C_DIS
LIN {X -0.229,Y -438.395,Z 457.474,A 0.000,B 0.000,C 90.000,E1 121.337} C_DIS
LIN {X -0.093,Y -434.835,Z 457.467,A 0.000,B 0.000,C 90.000,E1 120.001} C_DIS
LIN {X 0.030,Y -432.938,Z 457.463,A 0.000,B 0.000,C 90.000,E1 119.333} C_DIS
LIN {X -0.009,Y -432.938,Z 457.463,A 0.000,B 0.000,C 90.000,E1 119.333} C_DIS
LIN {X -0.098,Y -441.932,Z 457.444,A 0.000,B 0.000,C 90.000,E1 115.899} C_DIS
LIN {X 0.034,Y -444.846,Z 457.438,A 0.000,B 0.000,C 90.000,E1 114.899} C_DIS
LIN {X -0.130,Y -453.953,Z 457.417,A 0.000,B 0.000,C 90.000,E1 111.025} C_DIS
LIN {X 0.152,Y -457.428,Z 457.410,A 0.000,B 0.000,C 90.000,E1 109.704} C_DIS
LIN {X -0.194,Y -466.078,Z 457.387,A 0.000,B 0.000,C 90.000,E1 105.607} C_DIS
LIN {X -0.021,Y -467.647,Z 457.383,A 0.000,B 0.000,C 90.000,E1 104.954} C_DIS
LIN {X 0.174,Y -470.066,Z 457.374,A 0.000,B 0.000,C 90.000,E1 103.355} C_DIS
LIN {X -0.063,Y -475.867,Z 457.357,A 0.000,B 0.000,C 90.000,E1 100.254} C_DIS
LIN {X -0.225,Y -476.334,Z 457.355,A 0.000,B 0.000,C 90.000,E1 99.962} C_DIS
LIN {X -0.113,Y -480.144,Z 457.337,A 0.000,B 0.000,C 90.000,E1 96.720} C_DIS
LIN {X -0.178,Y -559.233,Z 457.337,A 0.000,B 0.000,C 90.000,E1 96.720} C_DIS
LIN {X 0.256,Y -563.077,Z 457.337,A 0.000,B 0.000,C 90.000,E1 96.663} C_DIS
LIN {X 0.255,Y -570.611,Z 457.337,A 0.000,B 0.000,C 90.000,E1 96.549} C_DIS
LIN {X 0.217,Y -577.047,Z 457.336,A 0.000,B 0.000,C 90.000,E1 96.429} C_DIS
LIN {X 0.189,Y -582.818,Z 457.335,A 0.000,B 0.000,C 90.000,E1 96.258} C_DIS
LIN {X 0.128,Y -588.948,Z 457.334,A 0.000,B 0.000,C 90.000,E1 96.030} C_DIS
LIN {X 0.241,Y -595.503,Z 457.332,A 0.000,B 0.000,C 90.000,E1 95.739} C_DIS
LIN {X 0.023,Y -601.509,Z 457.330,A 0.000,B 0.000,C 90.000,E1 95.454} C_DIS
LIN {X -0.064,Y -607.312,Z 457.328,A 0.000,B 0.000,C 90.000,E1 95.106} C_DIS
LIN {X -0.193,Y -611.507,Z 457.327,A 0.000,B 0.000,C 90.000,E1 94.821} C_DIS
LIN {X 0.038,Y -614.311,Z 457.326,A 0.000,B 0.000,C 90.000,E1 94.588} C_DIS
LIN {X -0.068,Y -620.665,Z 457.322,A 0.000,B 0.000,C 90.000,E1 94.012} C_DIS
LIN {X 0.201,Y -623.734,Z 457.320,A 0.000,B 0.000,C 90.000,E1 93.612} C_DIS
LIN {X -0.242,Y -626.536,Z 457.318,A 0.000,B 0.000,C 90.000,E1 93.269} C_DIS
LIN {X 0.276,Y -627.340,Z 457.317,A 0.000,B 0.000,C 90.000,E1 93.094} C_DIS
LIN {X -0.150,Y -629.086,Z 457.315,A 0.000,B 0.000,C 90.000,E1 92.751} C_DIS
LIN {X -0.074,Y -631.108,Z 457.312,A 0.000,B 0.000,C 90.000,E1 92.236} C_DIS
LIN {X 0.288,Y -632.044,Z 457.311,A 0.000,B 0.000,C 90.000,E1 91.949} C_DIS
LIN {X 0.040,Y -632.827,Z 457.310,A 0.000,B 0.000,C 90.000,E1 91.718} C_DIS
LIN {X 0.144,Y -633.764,Z 457.307,A 0.000,B 0.000,C 90.000,E1 91.203} C_DIS
LIN {X 0.258,Y -634.082,Z 457.304,A 0.000,B 0.000,C 90.000,E1 90.688} C_DIS
LIN {X -0.258,Y -634.095,Z 457.301,A 0.000,B 0.000,C 90.000,E1 90.229} C_DIS
LIN {X 0.119,Y -633.974,Z 457.300,A 0.000,B 0.000,C 90.000,E1 89.943} C_DIS
LIN {X 0.237,Y -633.336,Z 457.297,A 0.000,B 0.000,C 90.000,E1 89.427} C_DIS
LIN {X -0.022,Y -632.680,Z 457.296,A 0.000,B 0.000,C 90.000,E1 89.198} C_DIS
LIN {X 0.088,Y -630.941,Z 457.293,A 0.000,B 0.000,C 90.000,E1 88.682} C_DIS
LIN {X 0.203,Y -628.798,Z 457.290,A 0.000,B 0.000,C 90.000,E1 88.165} C_DIS
LIN {X 0.285,Y -626.305,Z 457.287,A 0.000,B 0.000,C 90.000,E1 87.650} C_DIS
LIN {X -0.062,Y -620.313,Z 457.282,A 0.000,B 0.000,C 90.000,E1 86.788} C_DIS
LIN {X 0.108,Y -617.129,Z 457.280,A 0.000,B 0.000,C 90.000,E1 86.388} C_DIS
LIN {X 0.255,Y -613.879,Z 457.278,A 0.000,B 0.000,C 90.000,E1 85.988} C_DIS
LIN {X -0.153,Y -609.995,Z 457.276,A 0.000,B 0.000,C 90.000,E1 85.641} C_DIS
LIN {X -0.312,Y -607.298,Z 457.274,A 0.000,B 0.000,C 90.000,E1 85.412} C_DIS
LIN {X -0.268,Y -601.473,Z 457.272,A 0.000,B 0.000,C 90.000,E1 84.951} C_DIS
LIN {X -0.181,Y -594.763,Z 457.270,A 0.000,B 0.000,C 90.000,E1 84.546} C_DIS
LIN {X -0.125,Y -587.934,Z 457.268,A 0.000,B 0.000,C 90.000,E1 84.204} C_DIS
LIN {X -0.223,Y -582.639,Z 457.266,A 0.000,B 0.000,C 90.000,E1 83.970} C_DIS
LIN {X 0.122,Y -576.526,Z 457.265,A 0.000,B 0.000,C 90.000,E1 83.742} C_DIS
LIN {X -0.247,Y -570.308,Z 457.265,A 0.000,B 0.000,C 90.000,E1 83.628} C_DIS
LIN {X 0.023,Y -564.808,Z 457.264,A 0.000,B 0.000,C 90.000,E1 83.514} C_DIS
LIN {X -0.228,Y -558.183,Z 457.264,A 0.000,B 0.000,C 90.000,E1 83.514} C_DIS
LIN {X -0.234,Y -484.995,Z 457.264,A 0.000,B 0.000,C 90.000,E1 83.514} C_DIS
LIN {X 0.241,Y -484.689,Z 457.254,A 0.000,B 0.000,C 90.000,E1 81.602} C_DIS
LIN {X -0.011,Y -483.031,Z 457.245,A 0.000,B 0.000,C 90.000,E1 80.095} C_DIS
LIN {X 0.140,Y -480.622,Z 457.228,A 0.000,B 0.000,C 90.000,E1 76.992} C_DIS
LIN {X -0.002,Y -480.290,Z 457.226,A 0.000,B 0.000,C 90.000,E1 76.700} C_DIS
LIN {X -0.097,Y -474.113,Z 457.200,A 0.000,B 0.000,C 90.000,E1 72.054} C_DIS
LIN {X -0.230,Y -465.571,Z 457.172,A 0.000,B 0.000,C 90.000,E1 67.050} C_DIS
LIN {X 0.045,Y -459.077,Z 457.155,A 0.000,B 0.000,C 90.000,E1 63.973} C_DIS
LIN {X 0.005,Y -459.087,Z 457.155,A 0.000,B 0.000,C 90.000,E1 63.973} C_DIS
LIN {X 0.115,Y -468.506,Z 457.148,A 0.000,B 0.000,C 90.000,E1 62.564} C_DIS
LIN {X -0.277,Y -475.868,Z 457.142,A 0.000,B 0.000,C 90.000,E1 61.513} C_DIS
LIN {X -0.128,Y -480.726,Z 457.137,A 0.000,B 0.000,C 90.000,E1 60.717} C_DIS
LIN {X -0.143,Y -483.501,Z 457.135,A 0.000,B 0.000,C 90.000,E1 60.255} C_DIS
LIN {X -0.145,Y -486.148,Z 457.132,A 0.000,B 0.000,C 90.000,E1 59.793} C_DIS
LIN {X 0.111,Y -490.024,Z 457.128,A 0.000,B 0.000,C 90.000,E1 58.997} C_DIS
LIN {X -0.064,Y -492.798,Z 457.124,A 0.000,B 0.000,C 90.000,E1 58.408} C_DIS
LIN {X -0.169,Y -495.796,Z 457.120,A 0.000,B 0.000,C 90.000,E1 57.661} C_DIS
LIN {X -0.045,Y -497.861,Z 457.117,A 0.000,B 0.000,C 90.000,E1 57.041} C_DIS
LIN {X 0.097,Y -499.482,Z 457.114,A 0.000,B 0.000,C 90.000,E1 56.421} C_DIS
LIN {X 0.129,Y -501.502,Z 457.109,A 0.000,B 0.000,C 90.000,E1 55.515} C_DIS
LIN {X 0.069,Y -503.178,Z 457.102,A 0.000,B 0.000,C 90.000,E1 54.322} C_DIS
LIN {X 0.252,Y -503.870,Z 457.099,A 0.000,B 0.000,C 90.000,E1 53.703} C_DIS
LIN {X -0.077,Y -504.439,Z 457.094,A 0.000,B 0.000,C 90.000,E1 52.844} C_DIS
LIN {X 0.307,Y -504.730,Z 457.089,A 0.000,B 0.000,C 90.000,E1 51.904} C_DIS
LIN {X -0.018,Y -504.861,Z 457.084,A 0.000,B 0.000,C 90.000,E1 51.045} C_DIS
LIN {X -0.027,Y -504.762,Z 457.079,A 0.000,B 0.000,C 90.000,E1 50.150} C_DIS
LIN {X -0.037,Y -504.455,Z 457.074,A 0.000,B 0.000,C 90.000,E1 49.256} C_DIS
LIN {X -0.114,Y -503.540,Z 457.064,A 0.000,B 0.000,C 90.000,E1 47.472} C_DIS
LIN {X -0.298,Y -502.767,Z 457.057,A 0.000,B 0.000,C 90.000,E1 46.296} C_DIS
LIN {X 0.071,Y -501.732,Z 457.049,A 0.000,B 0.000,C 90.000,E1 44.757} C_DIS
LIN {X -0.002,Y -501.053,Z 457.044,A 0.000,B 0.000,C 90.000,E1 43.866} C_DIS
LIN {X -0.152,Y -499.574,Z 457.034,A 0.000,B 0.000,C 90.000,E1 42.081} C_DIS
LIN {X 0.042,Y -498.058,Z 457.024,A 0.000,B 0.000,C 90.000,E1 40.253} C_DIS
LIN {X 0.009,Y -496.724,Z 457.015,A 0.000,B 0.000,C 90.000,E1 38.749} C_DIS
LIN {X 0.026,Y -495.339,Z 457.007,A 0.000,B 0.000,C 90.000,E1 37.237} C_DIS
LIN {X 0.018,Y -493.892,Z 456.999,A 0.000,B 0.000,C 90.000,E1 35.724} C_DIS
LIN {X 0.092,Y -492.206,Z 456.990,A 0.000,B 0.000,C 90.000,E1 34.199} C_DIS
LIN {X -0.118,Y -490.838,Z 456.983,A 0.000,B 0.000,C 90.000,E1 33.007} C_DIS
LIN {X -0.207,Y -489.389,Z 456.977,A 0.000,B 0.000,C 90.000,E1 31.799} C_DIS
LIN {X 0.166,Y -487.063,Z 456.966,A 0.000,B 0.000,C 90.000,E1 29.922} C_DIS
LIN {X 0.225,Y -484.349,Z 456.954,A 0.000,B 0.000,C 90.000,E1 27.769} C_DIS
LIN {X -0.012,Y -481.836,Z 456.943,A 0.000,B 0.000,C 90.000,E1 25.643} C_DIS
LIN {X 0.141,Y -479.357,Z 456.929,A 0.000,B 0.000,C 90.000,E1 23.153} C_DIS
LIN {X 0.244,Y -477.727,Z 456.917,A 0.000,B 0.000,C 90.000,E1 20.972} C_DIS
LIN {X -0.209,Y -476.304,Z 456.905,A 0.000,B 0.000,C 90.000,E1 18.852} C_DIS
LIN {X -0.038,Y -475.369,Z 456.896,A 0.000,B 0.000,C 90.000,E1 17.275} C_DIS
LIN {X -0.206,Y -474.102,Z 456.886,A 0.000,B 0.000,C 90.000,E1 15.426} C_DIS
LIN {X 0.162,Y -472.627,Z 456.872,A 0.000,B 0.000,C 90.000,E1 12.883} C_DIS
LIN {X -0.019,Y -471.739,Z 456.860,A 0.000,B 0.000,C 90.000,E1 10.715} C_DIS
LIN {X -0.107,Y -471.117,Z 456.846,A 0.000,B 0.000,C 90.000,E1 8.219} C_DIS
LIN {X -0.011,Y -471.139,Z 456.826,A 0.000,B 0.000,C 90.000,E1 4.759} C_DIS
LIN {X -0.017,Y -472.727,Z 456.804,A 0.000,B 0.000,C 90.000,E1 0.688} C_DIS
LIN {X -0.206,Y -474.225,Z 456.792,A 0.000,B 0.000,C 90.000,E1 358.568} C_DIS
LIN {X 0.038,Y -476.653,Z 456.778,A 0.000,B 0.000,C 90.000,E1 356.045} C_DIS
LIN {X 0.119,Y -480.435,Z 456.761,A 0.000,B 0.000,C 90.000,E1 352.932} C_DIS
LIN {X -0.064,Y -483.462,Z 456.749,A 0.000,B 0.000,C 90.000,E1 350.792} C_DIS
LIN {X 0.237,Y -485.858,Z 456.740,A 0.000,B 0.000,C 90.000,E1 349.218} C_DIS
LIN {X 0.033,Y -492.725,Z 456.720,A 0.000,B 0.000,C 90.000,E1 345.574} C_DIS
LIN {X 0.064,Y -497.408,Z 456.708,A 0.000,B 0.000,C 90.000,E1 343.449} C_DIS
LIN {X 0.170,Y -502.575,Z 456.696,A 0.000,B 0.000,C 90.000,E1 341.329} C_DIS
LIN {X -0.054,Y -507.895,Z 456.685,A 0.000,B 0.000,C 90.000,E1 339.263} C_DIS
LIN {X -0.199,Y -511.794,Z 456.677,A 0.000,B 0.000,C 90.000,E1 337.794} C_DIS
LIN {X -0.085,Y -515.647,Z 456.668,A 0.000,B 0.000,C 90.000,E1 336.305} C_DIS
LIN {X 0.173,Y -518.689,Z 456.662,A 0.000,B 0.000,C 90.000,E1 335.101} C_DIS
LIN {X -0.016,Y -523.998,Z 456.650,A 0.000,B 0.000,C 90.000,E1 333.076} C_DIS
LIN {X 0.240,Y -528.494,Z 456.641,A 0.000,B 0.000,C 90.000,E1 331.307} C_DIS
LIN {X -0.122,Y -533.068,Z 456.631,A 0.000,B 0.000,C 90.000,E1 329.616} C_DIS
LIN {X -0.303,Y -536.912,Z 456.623,A 0.000,B 0.000,C 90.000,E1 328.201} C_DIS
LIN {X 0.063,Y -542.271,Z 456.612,A 0.000,B 0.000,C 90.000,E1 326.167} C_DIS
LIN {X -0.107,Y -546.110,Z 456.604,A 0.000,B 0.000,C 90.000,E1 324.769} C_DIS
LIN {X 0.169,Y -550.844,Z 456.595,A 0.000,B 0.000,C 90.000,E1 323.050} C_DIS
LIN {X 0.118,Y -555.613,Z 456.586,A 0.000,B 0.000,C 90.000,E1 321.376} C_DIS
LIN {X -0.093,Y -562.088,Z 456.573,A 0.000,B 0.000,C 90.000,E1 319.175} C_DIS
LIN {X -0.033,Y -566.933,Z 456.564,A 0.000,B 0.000,C 90.000,E1 317.514} C_DIS
LIN {X 0.056,Y -570.840,Z 456.556,A 0.000,B 0.000,C 90.000,E1 316.134} C_DIS
LIN {X -0.097,Y -575.535,Z 456.547,A 0.000,B 0.000,C 90.000,E1 314.514} C_DIS
LIN {X 0.264,Y -580.269,Z 456.538,A 0.000,B 0.000,C 90.000,E1 312.852} C_DIS
LIN {X 0.161,Y -584.208,Z 456.531,A 0.000,B 0.000,C 90.000,E1 311.515} C_DIS
LIN {X 0.174,Y -588.161,Z 456.523,A 0.000,B 0.000,C 90.000,E1 310.172} C_DIS
LIN {X 0.056,Y -591.217,Z 456.517,A 0.000,B 0.000,C 90.000,E1 309.116} C_DIS
LIN {X -0.179,Y -594.904,Z 456.510,A 0.000,B 0.000,C 90.000,E1 307.810} C_DIS
LIN {X 0.128,Y -598.593,Z 456.503,A 0.000,B 0.000,C 90.000,E1 306.457} C_DIS
LIN {X 0.010,Y -602.131,Z 456.495,A 0.000,B 0.000,C 90.000,E1 305.152} C_DIS
LIN {X -0.169,Y -604.860,Z 456.490,A 0.000,B 0.000,C 90.000,E1 304.119} C_DIS
LIN {X 0.201,Y -607.482,Z 456.484,A 0.000,B 0.000,C 90.000,E1 303.038} C_DIS
LIN {X 0.047,Y -610.606,Z 456.476,A 0.000,B 0.000,C 90.000,E1 301.750} C_DIS
LIN {X -0.062,Y -613.586,Z 456.469,A 0.000,B 0.000,C 90.000,E1 300.463} C_DIS
LIN {X 0.074,Y -616.820,Z 456.461,A 0.000,B 0.000,C 90.000,E1 298.899} C_DIS
LIN {X -0.254,Y -619.498,Z 456.453,A 0.000,B 0.000,C 90.000,E1 297.641} C_DIS
LIN {X -0.283,Y -621.655,Z 456.448,A 0.000,B 0.000,C 90.000,E1 296.616} C_DIS
LIN {X -0.284,Y -623.117,Z 456.444,A 0.000,B 0.000,C 90.000,E1 295.848} C_DIS
LIN {X 0.308,Y -625.443,Z 456.436,A 0.000,B 0.000,C 90.000,E1 294.515} C_DIS
LIN {X -0.127,Y -627.915,Z 456.428,A 0.000,B 0.000,C 90.000,E1 293.025} C_DIS
LIN {X 0.076,Y -630.128,Z 456.419,A 0.000,B 0.000,C 90.000,E1 291.482} C_DIS
LIN {X 0.319,Y -632.161,Z 456.411,A 0.000,B 0.000,C 90.000,E1 289.939} C_DIS
LIN {X -0.238,Y -633.737,Z 456.404,A 0.000,B 0.000,C 90.000,E1 288.725} C_DIS
LIN {X -0.354,Y -635.404,Z 456.396,A 0.000,B 0.000,C 90.000,E1 287.221} C_DIS
LIN {X 0.340,Y -636.552,Z 456.389,A 0.000,B 0.000,C 90.000,E1 285.898} C_DIS
LIN {X -0.350,Y -637.326,Z 456.383,A 0.000,B 0.000,C 90.000,E1 284.954} C_DIS
LIN {X -0.253,Y -638.038,Z 456.377,A 0.000,B 0.000,C 90.000,E1 283.939} C_DIS
LIN {X 0.149,Y -638.628,Z 456.370,A 0.000,B 0.000,C 90.000,E1 282.647} C_DIS
LIN {X 0.138,Y -638.986,Z 456.366,A 0.000,B 0.000,C 90.000,E1 281.895} C_DIS
LIN {X -0.239,Y -639.360,Z 456.358,A 0.000,B 0.000,C 90.000,E1 280.423} C_DIS
LIN {X 0.225,Y -639.355,Z 456.352,A 0.000,B 0.000,C 90.000,E1 279.378} C_DIS
LIN {X -0.214,Y -639.201,Z 456.345,A 0.000,B 0.000,C 90.000,E1 278.163} C_DIS
LIN {X 0.163,Y -638.778,Z 456.340,A 0.000,B 0.000,C 90.000,E1 277.125} C_DIS
LIN {X -0.097,Y -638.123,Z 456.334,A 0.000,B 0.000,C 90.000,E1 276.144} C_DIS
LIN {X 0.267,Y -637.232,Z 456.329,A 0.000,B 0.000,C 90.000,E1 275.106} C_DIS
LIN {X -0.072,Y -635.987,Z 456.323,A 0.000,B 0.000,C 90.000,E1 274.131} C_DIS
LIN {X 0.246,Y -634.536,Z 456.317,A 0.000,B 0.000,C 90.000,E1 273.094} C_DIS
LIN {X -0.158,Y -632.877,Z 456.312,A 0.000,B 0.000,C 90.000,E1 272.121} C_DIS
LIN {X -0.191,Y -630.477,Z 456.305,A 0.000,B 0.000,C 90.000,E1 270.859} C_DIS
LIN {X -0.279,Y -627.895,Z 456.298,A 0.000,B 0.000,C 90.000,E1 269.599} C_DIS
LIN {X -0.132,Y -625.711,Z 456.292,A 0.000,B 0.000,C 90.000,E1 268.568} C_DIS
LIN {X -0.288,Y -622.751,Z 456.285,A 0.000,B 0.000,C 90.000,E1 267.306} C_DIS
LIN {X 0.125,Y -619.632,Z 456.278,A 0.000,B 0.000,C 90.000,E1 265.988} C_DIS
LIN {X 0.222,Y -617.108,Z 456.272,A 0.000,B 0.000,C 90.000,E1 264.951} C_DIS
LIN {X -0.033,Y -613.773,Z 456.265,A 0.000,B 0.000,C 90.000,E1 263.685} C_DIS
LIN {X -0.009,Y -611.100,Z 456.259,A 0.000,B 0.000,C 90.000,E1 262.648} C_DIS
LIN {X -0.297,Y -607.576,Z 456.252,A 0.000,B 0.000,C 90.000,E1 261.376} C_DIS
LIN {X -0.274,Y -604.779,Z 456.246,A 0.000,B 0.000,C 90.000,E1 260.330} C_DIS
LIN {X 0.021,Y -601.076,Z 456.239,A 0.000,B 0.000,C 90.000,E1 258.993} C_DIS
LIN {X -0.217,Y -595.706,Z 456.229,A 0.000,B 0.000,C 90.000,E1 257.173} C_DIS
LIN {X -0.242,Y -592.498,Z 456.223,A 0.000,B 0.000,C 90.000,E1 256.117} C_DIS
LIN {X 0.090,Y -588.484,Z 456.215,A 0.000,B 0.000,C 90.000,E1 254.755} C_DIS
LIN {X 0.106,Y -585.173,Z 456.209,A 0.000,B 0.000,C 90.000,E1 253.685} C_DIS
LIN {X 0.120,Y -580.127,Z 456.201,A 0.000,B 0.000,C 90.000,E1 252.072} C_DIS
LIN {X 0.185,Y -576.671,Z 456.195,A 0.000,B 0.000,C 90.000,E1 250.986} C_DIS
LIN {X 0.022,Y -572.267,Z 456.187,A 0.000,B 0.000,C 90.000,E1 249.645} C_DIS
LIN {X -0.193,Y -566.749,Z 456.178,A 0.000,B 0.000,C 90.000,E1 248.028} C_DIS
LIN {X 0.077,Y -563.865,Z 456.173,A 0.000,B 0.000,C 90.000,E1 247.177} C_DIS
LIN {X 0.011,Y -560.875,Z 456.169,A 0.000,B 0.000,C 90.000,E1 246.357} C_DIS
LIN {X 0.008,Y -555.807,Z 456.161,A 0.000,B 0.000,C 90.000,E1 244.973} C_DIS
LIN {X -0.091,Y -550.615,Z 456.153,A 0.000,B 0.000,C 90.000,E1 243.589} C_DIS
LIN {X 0.208,Y -545.323,Z 456.145,A 0.000,B 0.000,C 90.000,E1 242.153} C_DIS
LIN {X -0.116,Y -538.125,Z 456.134,A 0.000,B 0.000,C 90.000,E1 240.205} C_DIS
LIN {X -0.088,Y -530.979,Z 456.123,A 0.000,B 0.000,C 90.000,E1 238.201} C_DIS
LIN {X 0.033,Y -523.878,Z 456.112,A 0.000,B 0.000,C 90.000,E1 236.167} C_DIS
LIN {X -0.138,Y -519.791,Z 456.106,A 0.000,B 0.000,C 90.000,E1 235.022} C_DIS
LIN {X 0.002,Y -514.581,Z 456.098,A 0.000,B 0.000,C 90.000,E1 233.543} C_DIS
LIN {X -0.133,Y -502.114,Z 456.076,A 0.000,B 0.000,C 90.000,E1 229.703} C_DIS
LIN {X -0.090,Y -495.878,Z 456.064,A 0.000,B 0.000,C 90.000,E1 227.595} C_DIS
LIN {X -0.032,Y -489.002,Z 456.051,A 0.000,B 0.000,C 90.000,E1 225.162} C_DIS
LIN {X 0.204,Y -484.074,Z 456.041,A 0.000,B 0.000,C 90.000,E1 223.299} C_DIS
LIN {X 0.020,Y -479.239,Z 456.030,A 0.000,B 0.000,C 90.000,E1 221.472} C_DIS
LIN {X -0.014,Y -473.196,Z 456.017,A 0.000,B 0.000,C 90.000,E1 218.991} C_DIS
LIN {X 0.059,Y -468.147,Z 456.004,A 0.000,B 0.000,C 90.000,E1 216.790} C_DIS
LIN {X 0.056,Y -464.095,Z 455.994,A 0.000,B 0.000,C 90.000,E1 214.898} C_DIS
LIN {X 0.202,Y -458.858,Z 455.980,A 0.000,B 0.000,C 90.000,E1 212.339} C_DIS
LIN {X -0.026,Y -454.462,Z 455.967,A 0.000,B 0.000,C 90.000,E1 210.129} C_DIS
LIN {X 0.107,Y -450.655,Z 455.957,A 0.000,B 0.000,C 90.000,E1 208.180} C_DIS
LIN {X 0.088,Y -447.553,Z 455.948,A 0.000,B 0.000,C 90.000,E1 206.565} C_DIS
LIN {X 0.119,Y -443.039,Z 455.935,A 0.000,B 0.000,C 90.000,E1 204.283} C_DIS
LIN {X -0.162,Y -438.463,Z 455.922,A 0.000,B 0.000,C 90.000,E1 202.025} C_DIS
LIN {X 0.065,Y -434.125,Z 455.909,A 0.000,B 0.000,C 90.000,E1 199.685} C_DIS
LIN {X 0.151,Y -430.016,Z 455.897,A 0.000,B 0.000,C 90.000,E1 197.347} C_DIS
LIN {X -0.195,Y -425.808,Z 455.882,A 0.000,B 0.000,C 90.000,E1 194.717} C_DIS
LIN {X -0.145,Y -422.417,Z 455.869,A 0.000,B 0.000,C 90.000,E1 192.355} C_DIS
LIN {X 0.104,Y -418.934,Z 455.854,A 0.000,B 0.000,C 90.000,E1 189.613} C_DIS
LIN {X 0.105,Y -415.423,Z 455.837,A 0.000,B 0.000,C 90.000,E1 186.549} C_DIS
LIN {X -0.135,Y -412.905,Z 455.823,A 0.000,B 0.000,C 90.000,E1 184.188} C_DIS
LIN {X -0.081,Y -410.494,Z 455.808,A 0.000,B 0.000,C 90.000,E1 181.432} C_DIS
LIN {X -0.169,Y -408.161,Z 455.787,A 0.000,B 0.000,C 90.000,E1 177.650} C_DIS
LIN {X 0.182,Y -407.256,Z 455.773,A 0.000,B 0.000,C 90.000,E1 175.179} C_DIS
LIN {X 0.122,Y -406.983,Z 455.754,A 0.000,B 0.000,C 90.000,E1 171.724} C_DIS
LIN {X -0.192,Y -407.303,Z 455.743,A 0.000,B 0.000,C 90.000,E1 169.690} C_DIS
LIN {X -0.177,Y -408.639,Z 455.723,A 0.000,B 0.000,C 90.000,E1 166.228} C_DIS
LIN {X -0.185,Y -409.787,Z 455.712,A 0.000,B 0.000,C 90.000,E1 164.157} C_DIS
LIN {X 0.073,Y -412.473,Z 455.693,A 0.000,B 0.000,C 90.000,E1 160.678} C_DIS
LIN {X -0.117,Y -414.500,Z 455.681,A 0.000,B 0.000,C 90.000,E1 158.646} C_DIS
LIN {X -0.183,Y -417.661,Z 455.666,A 0.000,B 0.000,C 90.000,E1 155.921} C_DIS
LIN {X -0.012,Y -421.195,Z 455.651,A 0.000,B 0.000,C 90.000,E1 153.179} C_DIS
LIN {X 0.094,Y -425.003,Z 455.636,A 0.000,B 0.000,C 90.000,E1 150.461} C_DIS
LIN {X 0.007,Y -427.900,Z 455.625,A 0.000,B 0.000,C 90.000,E1 148.456} C_DIS
LIN {X 0.218,Y -431.019,Z 455.614,A 0.000,B 0.000,C 90.000,E1 146.421} C_DIS
LIN {X -0.221,Y -434.315,Z 455.603,A 0.000,B 0.000,C 90.000,E1 144.482} C_DIS
LIN {X -0.131,Y -438.863,Z 455.588,A 0.000,B 0.000,C 90.000,E1 141.823} C_DIS
LIN {X 0.013,Y -443.044,Z 455.575,A 0.000,B 0.000,C 90.000,E1 139.504} C_DIS
LIN {X -0.065,Y -447.259,Z 455.562,A 0.000,B 0.000,C 90.000,E1 137.229} C_DIS
LIN {X 0.236,Y -449.451,Z 455.555,A 0.000,B 0.000,C 90.000,E1 135.891} C_DIS
LIN {X 0.242,Y -450.904,Z 455.550,A 0.000,B 0.000,C 90.000,E1 134.919} C_DIS
LIN {X -0.036,Y -452.500,Z 455.543,A 0.000,B 0.000,C 90.000,E1 133.662} C_DIS
LIN {X 0.004,Y -453.512,Z 455.537,A 0.000,B 0.000,C 90.000,E1 132.690} C_DIS
LIN {X -0.256,Y -454.216,Z 455.532,A 0.000,B 0.000,C 90.000,E1 131.757} C_DIS
LIN {X 0.114,Y -454.580,Z 455.528,A 0.000,B 0.000,C 90.000,E1 131.067} C_DIS
LIN {X 0.207,Y -454.746,Z 455.523,A 0.000,B 0.000,C 90.000,E1 130.092} C_DIS
LIN {X 0.013,Y -454.474,Z 455.518,A 0.000,B 0.000,C 90.000,E1 129.152} C_DIS
LIN {X 0.103,Y -453.768,Z 455.512,A 0.000,B 0.000,C 90.000,E1 128.177} C_DIS
LIN {X -0.098,Y -452.690,Z 455.507,A 0.000,B 0.000,C 90.000,E1 127.237} C_DIS
LIN {X 0.053,Y -451.399,Z 455.501,A 0.000,B 0.000,C 90.000,E1 126.251} C_DIS
LIN {X -0.176,Y -449.752,Z 455.496,A 0.000,B 0.000,C 90.000,E1 125.311} C_DIS
LIN {X -0.062,Y -447.772,Z 455.491,A 0.000,B 0.000,C 90.000,E1 124.326} C_DIS
LIN {X -0.223,Y -445.470,Z 455.485,A 0.000,B 0.000,C 90.000,E1 123.372} C_DIS
LIN {X 0.261,Y -442.092,Z 455.478,A 0.000,B 0.000,C 90.000,E1 122.005} C_DIS
LIN {X 0.076,Y -438.547,Z 455.471,A 0.000,B 0.000,C 90.000,E1 120.718} C_DIS
LIN {X -0.009,Y -434.740,Z 455.463,A 0.000,B 0.000,C 90.000,E1 119.411} C_DIS
LIN {X 0.080,Y -433.650,Z 455.461,A 0.000,B 0.000,C 90.000,E1 119.027} C_DIS
LIN {X 0.041,Y -433.642,Z 455.461,A 0.000,B 0.000,C 90.000,E1 119.027} C_DIS
LIN {X -0.123,Y -443.224,Z 455.441,A 0.000,B 0.000,C 90.000,E1 115.463} C_DIS
LIN {X 0.171,Y -445.082,Z 455.438,A 0.000,B 0.000,C 90.000,E1 114.771} C_DIS
LIN {X -0.145,Y -454.244,Z 455.416,A 0.000,B 0.000,C 90.000,E1 110.918} C_DIS
LIN {X -0.029,Y -456.907,Z 455.411,A 0.000,B 0.000,C 90.000,E1 109.939} C_DIS
LIN {X -0.128,Y -457.620,Z 455.409,A 0.000,B 0.000,C 90.000,E1 109.631} C_DIS
LIN {X -0.041,Y -466.339,Z 455.386,A 0.000,B 0.000,C 90.000,E1 105.481} C_DIS
LIN {X 0.132,Y -467.874,Z 455.383,A 0.000,B 0.000,C 90.000,E1 104.828} C_DIS
LIN {X 0.161,Y -475.435,Z 455.358,A 0.000,B 0.000,C 90.000,E1 100.433} C_DIS
LIN {X -0.001,Y -476.085,Z 455.356,A 0.000,B 0.000,C 90.000,E1 100.141} C_DIS
LIN {X 0.116,Y -481.040,Z 455.334,A 0.000,B 0.000,C 90.000,E1 96.087} C_DIS
LIN {X 0.088,Y -564.836,Z 455.334,A 0.000,B 0.000,C 90.000,E1 96.087} C_DIS
LIN {X -0.051,Y -568.412,Z 455.334,A 0.000,B 0.000,C 90.000,E1 96.087} C_DIS
LIN {X -0.017,Y -575.023,Z 455.333,A 0.000,B 0.000,C 90.000,E1 95.967} C_DIS
LIN {X 0.071,Y -579.390,Z 455.333,A 0.000,B 0.000,C 90.000,E1 95.853} C_DIS
LIN {X 0.003,Y -581.787,Z 455.332,A 0.000,B 0.000,C 90.000,E1 95.796} C_DIS
LIN {X 0.217,Y -587.901,Z 455.331,A 0.000,B 0.000,C 90.000,E1 95.568} C_DIS
LIN {X -0.153,Y -594.001,Z 455.330,A 0.000,B 0.000,C 90.000,E1 95.334} C_DIS
LIN {X 0.266,Y -600.214,Z 455.328,A 0.000,B 0.000,C 90.000,E1 94.992} C_DIS
LIN {X 0.282,Y -606.024,Z 455.326,A 0.000,B 0.000,C 90.000,E1 94.645} C_DIS
LIN {X 0.293,Y -610.190,Z 455.324,A 0.000,B 0.000,C 90.000,E1 94.359} C_DIS
LIN {X -0.009,Y -614.183,Z 455.323,A 0.000,B 0.000,C 90.000,E1 94.073} C_DIS
LIN {X -0.090,Y -619.255,Z 455.320,A 0.000,B 0.000,C 90.000,E1 93.612} C_DIS
LIN {X -0.193,Y -620.312,Z 455.319,A 0.000,B 0.000,C 90.000,E1 93.498} C_DIS
LIN {X 0.058,Y -623.016,Z 455.317,A 0.000,B 0.000,C 90.000,E1 93.094} C_DIS
LIN {X 0.093,Y -626.000,Z 455.314,A 0.000,B 0.000,C 90.000,E1 92.579} C_DIS
LIN {X -0.193,Y -627.097,Z 455.313,A 0.000,B 0.000,C 90.000,E1 92.350} C_DIS
LIN {X -0.128,Y -628.748,Z 455.310,A 0.000,B 0.000,C 90.000,E1 91.835} C_DIS
LIN {X -0.032,Y -629.837,Z 455.307,A 0.000,B 0.000,C 90.000,E1 91.318} C_DIS
LIN {X 0.054,Y -630.391,Z 455.305,A 0.000,B 0.000,C 90.000,E1 90.802} C_DIS
LIN {X -0.215,Y -630.540,Z 455.303,A 0.000,B 0.000,C 90.000,E1 90.573} C_DIS
LIN {X -0.121,Y -630.446,Z 455.300,A 0.000,B 0.000,C 90.000,E1 90.057} C_DIS
LIN {X -0.027,Y -629.539,Z 455.297,A 0.000,B 0.000,C 90.000,E1 89.542} C_DIS
LIN {X -0.211,Y -627.319,Z 455.293,A 0.000,B 0.000,C 90.000,E1 88.797} C_DIS
LIN {X -0.139,Y -625.219,Z 455.290,A 0.000,B 0.000,C 90.000,E1 88.282} C_DIS
LIN {X 0.268,Y -620.610,Z 455.286,A 0.000,B 0.000,C 90.000,E1 87.478} C_DIS
LIN {X -0.180,Y -618.009,Z 455.284,A 0.000,B 0.000,C 90.000,E1 87.135} C_DIS
LIN {X -0.145,Y -613.905,Z 455.281,A 0.000,B 0.000,C 90.000,E1 86.617} C_DIS
LIN {X -0.297,Y -607.879,Z 455.278,A 0.000,B 0.000,C 90.000,E1 85.988} C_DIS
LIN {X 0.041,Y -604.720,Z 455.276,A 0.000,B 0.000,C 90.000,E1 85.698} C_DIS
LIN {X 0.133,Y -601.836,Z 455.275,A 0.000,B 0.000,C 90.000,E1 85.469} C_DIS
LIN {X -0.084,Y -596.774,Z 455.273,A 0.000,B 0.000,C 90.000,E1 85.179} C_DIS
LIN {X -0.219,Y -593.354,Z 455.272,A 0.000,B 0.000,C 90.000,E1 85.008} C_DIS
LIN {X -0.035,Y -586.313,Z 455.270,A 0.000,B 0.000,C 90.000,E1 84.666} C_DIS
LIN {X 0.232,Y -582.834,Z 455.270,A 0.000,B 0.000,C 90.000,E1 84.489} C_DIS
LIN {X 0.046,Y -576.944,Z 455.268,A 0.000,B 0.000,C 90.000,E1 84.318} C_DIS
LIN {X -0.257,Y -569.942,Z 455.268,A 0.000,B 0.000,C 90.000,E1 84.204} C_DIS
LIN {X -0.008,Y -563.919,Z 455.267,A 0.000,B 0.000,C 90.000,E1 84.090} C_DIS
LIN {X -0.055,Y -485.205,Z 455.267,A 0.000,B 0.000,C 90.000,E1 84.090} C_DIS
LIN {X -0.221,Y -484.674,Z 455.253,A 0.000,B 0.000,C 90.000,E1 81.602} C_DIS
LIN {X 0.148,Y -480.592,Z 455.228,A 0.000,B 0.000,C 90.000,E1 76.937} C_DIS
LIN {X -0.139,Y -479.685,Z 455.224,A 0.000,B 0.000,C 90.000,E1 76.353} C_DIS
LIN {X -0.105,Y -474.027,Z 455.200,A 0.000,B 0.000,C 90.000,E1 72.000} C_DIS
LIN {X -0.018,Y -465.947,Z 455.174,A 0.000,B 0.000,C 90.000,E1 67.283} C_DIS
LIN {X -0.075,Y -465.446,Z 455.172,A 0.000,B 0.000,C 90.000,E1 66.975} C_DIS
LIN {X -0.027,Y -459.501,Z 455.157,A 0.000,B 0.000,C 90.000,E1 64.204} C_DIS
LIN {X -0.068,Y -459.522,Z 455.157,A 0.000,B 0.000,C 90.000,E1 64.204} C_DIS
LIN {X -0.250,Y -468.785,Z 455.149,A 0.000,B 0.000,C 90.000,E1 62.871} C_DIS
LIN {X 0.012,Y -475.217,Z 455.144,A 0.000,B 0.000,C 90.000,E1 61.897} C_DIS
LIN {X -0.038,Y -481.197,Z 455.139,A 0.000,B 0.000,C 90.000,E1 60.973} C_DIS
LIN {X 0.150,Y -484.914,Z 455.135,A 0.000,B 0.000,C 90.000,E1 60.333} C_DIS
LIN {X -0.058,Y -488.344,Z 455.132,A 0.000,B 0.000,C 90.000,E1 59.744} C_DIS
LIN {X 0.005,Y -491.468,Z 455.129,A 0.000,B 0.000,C 90.000,E1 59.125} C_DIS
LIN {X -0.159,Y -494.274,Z 455.125,A 0.000,B 0.000,C 90.000,E1 58.535} C_DIS
LIN {X -0.044,Y -496.730,Z 455.122,A 0.000,B 0.000,C 90.000,E1 57.916} C_DIS
LIN {X -0.177,Y -498.807,Z 455.118,A 0.000,B 0.000,C 90.000,E1 57.327} C_DIS
LIN {X -0.030,Y -500.550,Z 455.115,A 0.000,B 0.000,C 90.000,E1 56.707} C_DIS
LIN {X -0.158,Y -501.373,Z 455.113,A 0.000,B 0.000,C 90.000,E1 56.421} C_DIS
LIN {X -0.106,Y -503.257,Z 455.108,A 0.000,B 0.000,C 90.000,E1 55.515} C_DIS
LIN {X -0.031,Y -504.511,Z 455.103,A 0.000,B 0.000,C 90.000,E1 54.609} C_DIS
LIN {X 0.162,Y -505.283,Z 455.100,A 0.000,B 0.000,C 90.000,E1 53.989} C_DIS
LIN {X -0.153,Y -505.886,Z 455.095,A 0.000,B 0.000,C 90.000,E1 53.130} C_DIS
LIN {X 0.146,Y -506.232,Z 455.089,A 0.000,B 0.000,C 90.000,E1 51.904} C_DIS
LIN {X -0.060,Y -506.336,Z 455.085,A 0.000,B 0.000,C 90.000,E1 51.331} C_DIS
LIN {X -0.051,Y -506.238,Z 455.080,A 0.000,B 0.000,C 90.000,E1 50.436} C_DIS
LIN {X -0.042,Y -505.937,Z 455.075,A 0.000,B 0.000,C 90.000,E1 49.542} C_DIS
LIN {X -0.083,Y -504.965,Z 455.065,A 0.000,B 0.000,C 90.000,E1 47.757} C_DIS
LIN {X 0.125,Y -504.148,Z 455.059,A 0.000,B 0.000,C 90.000,E1 46.539} C_DIS
LIN {X -0.193,Y -503.042,Z 455.050,A 0.000,B 0.000,C 90.000,E1 45.081} C_DIS
LIN {X -0.034,Y -502.086,Z 455.044,A 0.000,B 0.000,C 90.000,E1 43.866} C_DIS
LIN {X -0.162,Y -500.570,Z 455.034,A 0.000,B 0.000,C 90.000,E1 42.081} C_DIS
LIN {X 0.054,Y -499.043,Z 455.024,A 0.000,B 0.000,C 90.000,E1 40.253} C_DIS
LIN {X 0.040,Y -497.687,Z 455.015,A 0.000,B 0.000,C 90.000,E1 38.749} C_DIS
LIN {X 0.075,Y -496.286,Z 455.007,A 0.000,B 0.000,C 90.000,E1 37.237} C_DIS
LIN {X 0.223,Y -495.109,Z 455.000,A 0.000,B 0.000,C 90.000,E1 36.011} C_DIS
LIN {X 0.060,Y -493.820,Z 454.994,A 0.000,B 0.000,C 90.000,E1 34.818} C_DIS
LIN {X -0.023,Y -491.737,Z 454.983,A 0.000,B 0.000,C 90.000,E1 33.007} C_DIS
LIN {X -0.098,Y -490.243,Z 454.977,A 0.000,B 0.000,C 90.000,E1 31.799} C_DIS
LIN {X 0.051,Y -487.907,Z 454.966,A 0.000,B 0.000,C 90.000,E1 29.951} C_DIS
LIN {X 0.108,Y -486.698,Z 454.961,A 0.000,B 0.000,C 90.000,E1 29.027} C_DIS
LIN {X 0.168,Y -484.099,Z 454.949,A 0.000,B 0.000,C 90.000,E1 26.873} C_DIS
LIN {X -0.286,Y -481.351,Z 454.936,A 0.000,B 0.000,C 90.000,E1 24.463} C_DIS
LIN {X -0.159,Y -478.527,Z 454.917,A 0.000,B 0.000,C 90.000,E1 21.046} C_DIS
LIN {X 0.005,Y -476.902,Z 454.903,A 0.000,B 0.000,C 90.000,E1 18.544} C_DIS
LIN {X 0.213,Y -476.155,Z 454.896,A 0.000,B 0.000,C 90.000,E1 17.275} C_DIS
LIN {X 0.061,Y -474.864,Z 454.886,A 0.000,B 0.000,C 90.000,E1 15.426} C_DIS
LIN {X 0.050,Y -473.537,Z 454.874,A 0.000,B 0.000,C 90.000,E1 13.244} C_DIS
LIN {X -0.137,Y -472.254,Z 454.856,A 0.000,B 0.000,C 90.000,E1 10.141} C_DIS
LIN {X 0.223,Y -471.812,Z 454.846,A 0.000,B 0.000,C 90.000,E1 8.219} C_DIS
LIN {X 0.119,Y -471.830,Z 454.825,A 0.000,B 0.000,C 90.000,E1 4.473} C_DIS
LIN {X 0.159,Y -473.505,Z 454.802,A 0.000,B 0.000,C 90.000,E1 0.401} C_DIS
LIN {X -0.130,Y -475.359,Z 454.788,A 0.000,B 0.000,C 90.000,E1 357.936} C_DIS
LIN {X -0.110,Y -477.602,Z 454.776,A 0.000,B 0.000,C 90.000,E1 355.755} C_DIS
LIN {X 0.171,Y -481.060,Z 454.761,A 0.000,B 0.000,C 90.000,E1 352.932} C_DIS
LIN {X 0.003,Y -484.083,Z 454.749,A 0.000,B 0.000,C 90.000,E1 350.792} C_DIS
LIN {X -0.161,Y -486.478,Z 454.740,A 0.000,B 0.000,C 90.000,E1 349.275} C_DIS
LIN {X 0.039,Y -494.023,Z 454.718,A 0.000,B 0.000,C 90.000,E1 345.283} C_DIS
LIN {X 0.173,Y -501.744,Z 454.700,A 0.000,B 0.000,C 90.000,E1 341.945} C_DIS
LIN {X -0.080,Y -507.022,Z 454.688,A 0.000,B 0.000,C 90.000,E1 339.880} C_DIS
LIN {X -0.132,Y -511.718,Z 454.678,A 0.000,B 0.000,C 90.000,E1 338.103} C_DIS
LIN {X -0.019,Y -515.645,Z 454.670,A 0.000,B 0.000,C 90.000,E1 336.613} C_DIS
LIN {X -0.092,Y -519.471,Z 454.662,A 0.000,B 0.000,C 90.000,E1 335.153} C_DIS
LIN {X -0.256,Y -524.809,Z 454.651,A 0.000,B 0.000,C 90.000,E1 333.127} C_DIS
LIN {X -0.230,Y -529.388,Z 454.641,A 0.000,B 0.000,C 90.000,E1 331.385} C_DIS
LIN {X 0.126,Y -534.782,Z 454.630,A 0.000,B 0.000,C 90.000,E1 329.331} C_DIS
LIN {X -0.016,Y -538.639,Z 454.622,A 0.000,B 0.000,C 90.000,E1 327.916} C_DIS
LIN {X -0.046,Y -544.048,Z 454.611,A 0.000,B 0.000,C 90.000,E1 325.928} C_DIS
LIN {X 0.272,Y -547.911,Z 454.603,A 0.000,B 0.000,C 90.000,E1 324.482} C_DIS
LIN {X -0.180,Y -552.687,Z 454.594,A 0.000,B 0.000,C 90.000,E1 322.844} C_DIS
LIN {X -0.198,Y -557.476,Z 454.584,A 0.000,B 0.000,C 90.000,E1 321.170} C_DIS
LIN {X -0.094,Y -563.251,Z 454.573,A 0.000,B 0.000,C 90.000,E1 319.218} C_DIS
LIN {X 0.038,Y -568.159,Z 454.564,A 0.000,B 0.000,C 90.000,E1 317.553} C_DIS
LIN {X -0.274,Y -572.122,Z 454.557,A 0.000,B 0.000,C 90.000,E1 316.215} C_DIS
LIN {X 0.129,Y -577.657,Z 454.546,A 0.000,B 0.000,C 90.000,E1 314.271} C_DIS
LIN {X -0.286,Y -582.459,Z 454.537,A 0.000,B 0.000,C 90.000,E1 312.690} C_DIS
LIN {X -0.095,Y -585.685,Z 454.531,A 0.000,B 0.000,C 90.000,E1 311.595} C_DIS
LIN {X -0.055,Y -589.647,Z 454.524,A 0.000,B 0.000,C 90.000,E1 310.253} C_DIS
LIN {X -0.152,Y -592.752,Z 454.518,A 0.000,B 0.000,C 90.000,E1 309.197} C_DIS
LIN {X 0.006,Y -596.451,Z 454.510,A 0.000,B 0.000,C 90.000,E1 307.855} C_DIS
LIN {X -0.025,Y -600.203,Z 454.503,A 0.000,B 0.000,C 90.000,E1 306.537} C_DIS
LIN {X -0.112,Y -603.748,Z 454.496,A 0.000,B 0.000,C 90.000,E1 305.231} C_DIS
LIN {X -0.267,Y -606.504,Z 454.490,A 0.000,B 0.000,C 90.000,E1 304.199} C_DIS
LIN {X -0.383,Y -609.160,Z 454.484,A 0.000,B 0.000,C 90.000,E1 303.166} C_DIS
LIN {X 0.328,Y -612.321,Z 454.477,A 0.000,B 0.000,C 90.000,E1 301.799} C_DIS
LIN {X 0.213,Y -615.890,Z 454.468,A 0.000,B 0.000,C 90.000,E1 300.256} C_DIS
LIN {X -0.148,Y -619.155,Z 454.460,A 0.000,B 0.000,C 90.000,E1 298.743} C_DIS
LIN {X -0.184,Y -621.317,Z 454.454,A 0.000,B 0.000,C 90.000,E1 297.719} C_DIS
LIN {X 0.098,Y -623.484,Z 454.448,A 0.000,B 0.000,C 90.000,E1 296.668} C_DIS
LIN {X -0.127,Y -626.454,Z 454.440,A 0.000,B 0.000,C 90.000,E1 295.155} C_DIS
LIN {X -0.068,Y -628.212,Z 454.434,A 0.000,B 0.000,C 90.000,E1 294.131} C_DIS
LIN {X 0.105,Y -630.261,Z 454.427,A 0.000,B 0.000,C 90.000,E1 292.845} C_DIS
LIN {X -0.019,Y -632.128,Z 454.420,A 0.000,B 0.000,C 90.000,E1 291.589} C_DIS
LIN {X 0.232,Y -633.905,Z 454.413,A 0.000,B 0.000,C 90.000,E1 290.301} C_DIS
LIN {X -0.299,Y -635.554,Z 454.406,A 0.000,B 0.000,C 90.000,E1 289.087} C_DIS
LIN {X -0.203,Y -636.946,Z 454.399,A 0.000,B 0.000,C 90.000,E1 287.819} C_DIS
LIN {X -0.090,Y -638.277,Z 454.392,A 0.000,B 0.000,C 90.000,E1 286.551} C_DIS
LIN {X 0.307,Y -639.479,Z 454.384,A 0.000,B 0.000,C 90.000,E1 285.009} C_DIS
LIN {X 0.116,Y -640.355,Z 454.377,A 0.000,B 0.000,C 90.000,E1 283.772} C_DIS
LIN {X 0.249,Y -641.173,Z 454.367,A 0.000,B 0.000,C 90.000,E1 282.007} C_DIS
LIN {X -0.208,Y -641.555,Z 454.359,A 0.000,B 0.000,C 90.000,E1 280.546} C_DIS
LIN {X -0.176,Y -641.639,Z 454.354,A 0.000,B 0.000,C 90.000,E1 279.792} C_DIS
LIN {X 0.163,Y -641.489,Z 454.347,A 0.000,B 0.000,C 90.000,E1 278.511} C_DIS
LIN {X -0.064,Y -641.220,Z 454.342,A 0.000,B 0.000,C 90.000,E1 277.530} C_DIS
LIN {X 0.164,Y -640.448,Z 454.335,A 0.000,B 0.000,C 90.000,E1 276.258} C_DIS
LIN {X -0.079,Y -639.558,Z 454.329,A 0.000,B 0.000,C 90.000,E1 275.277} C_DIS
LIN {X 0.245,Y -638.327,Z 454.324,A 0.000,B 0.000,C 90.000,E1 274.245} C_DIS
LIN {X 0.174,Y -637.280,Z 454.320,A 0.000,B 0.000,C 90.000,E1 273.498} C_DIS
LIN {X 0.218,Y -635.195,Z 454.313,A 0.000,B 0.000,C 90.000,E1 272.236} C_DIS
LIN {X 0.222,Y -632.808,Z 454.306,A 0.000,B 0.000,C 90.000,E1 270.974} C_DIS
LIN {X 0.170,Y -630.202,Z 454.299,A 0.000,B 0.000,C 90.000,E1 269.714} C_DIS
LIN {X -0.280,Y -628.018,Z 454.293,A 0.000,B 0.000,C 90.000,E1 268.740} C_DIS
LIN {X -0.057,Y -624.415,Z 454.284,A 0.000,B 0.000,C 90.000,E1 267.192} C_DIS
LIN {X -0.194,Y -621.253,Z 454.277,A 0.000,B 0.000,C 90.000,E1 265.927} C_DIS
LIN {X 0.187,Y -617.995,Z 454.270,A 0.000,B 0.000,C 90.000,E1 264.609} C_DIS
LIN {X -0.320,Y -613.973,Z 454.262,A 0.000,B 0.000,C 90.000,E1 263.109} C_DIS
LIN {X 0.046,Y -610.477,Z 454.254,A 0.000,B 0.000,C 90.000,E1 261.781} C_DIS
LIN {X 0.175,Y -606.196,Z 454.246,A 0.000,B 0.000,C 90.000,E1 260.208} C_DIS
LIN {X -0.091,Y -602.442,Z 454.238,A 0.000,B 0.000,C 90.000,E1 258.926} C_DIS
LIN {X -0.127,Y -597.816,Z 454.230,A 0.000,B 0.000,C 90.000,E1 257.353} C_DIS
LIN {X 0.015,Y -594.606,Z 454.224,A 0.000,B 0.000,C 90.000,E1 256.284} C_DIS
LIN {X -0.027,Y -591.382,Z 454.218,A 0.000,B 0.000,C 90.000,E1 255.227} C_DIS
LIN {X -0.283,Y -587.253,Z 454.211,A 0.000,B 0.000,C 90.000,E1 253.921} C_DIS
LIN {X -0.219,Y -582.149,Z 454.202,A 0.000,B 0.000,C 90.000,E1 252.308} C_DIS
LIN {X 0.263,Y -577.794,Z 454.194,A 0.000,B 0.000,C 90.000,E1 250.913} C_DIS
LIN {X 0.128,Y -573.326,Z 454.187,A 0.000,B 0.000,C 90.000,E1 249.571} C_DIS
LIN {X -0.089,Y -568.732,Z 454.179,A 0.000,B 0.000,C 90.000,E1 248.230} C_DIS
LIN {X 0.228,Y -564.856,Z 454.173,A 0.000,B 0.000,C 90.000,E1 247.102} C_DIS
LIN {X -0.246,Y -560.825,Z 454.167,A 0.000,B 0.000,C 90.000,E1 246.049} C_DIS
LIN {X -0.251,Y -555.691,Z 454.159,A 0.000,B 0.000,C 90.000,E1 244.665} C_DIS
LIN {X -0.108,Y -550.479,Z 454.151,A 0.000,B 0.000,C 90.000,E1 243.256} C_DIS
LIN {X 0.175,Y -543.049,Z 454.140,A 0.000,B 0.000,C 90.000,E1 241.257} C_DIS
LIN {X -0.133,Y -537.925,Z 454.133,A 0.000,B 0.000,C 90.000,E1 239.871} C_DIS
LIN {X 0.189,Y -531.784,Z 454.123,A 0.000,B 0.000,C 90.000,E1 238.122} C_DIS
LIN {X -0.104,Y -524.647,Z 454.112,A 0.000,B 0.000,C 90.000,E1 236.135} C_DIS
LIN {X -0.174,Y -519.503,Z 454.104,A 0.000,B 0.000,C 90.000,E1 234.689} C_DIS
LIN {X 0.019,Y -515.337,Z 454.097,A 0.000,B 0.000,C 90.000,E1 233.497} C_DIS
LIN {X -0.159,Y -502.903,Z 454.076,A 0.000,B 0.000,C 90.000,E1 229.666} C_DIS
LIN {X -0.050,Y -496.651,Z 454.064,A 0.000,B 0.000,C 90.000,E1 227.553} C_DIS
LIN {X 0.016,Y -489.785,Z 454.051,A 0.000,B 0.000,C 90.000,E1 225.121} C_DIS
LIN {X -0.074,Y -484.869,Z 454.041,A 0.000,B 0.000,C 90.000,E1 223.299} C_DIS
LIN {X 0.080,Y -480.013,Z 454.030,A 0.000,B 0.000,C 90.000,E1 221.434} C_DIS
LIN {X -0.038,Y -474.700,Z 454.018,A 0.000,B 0.000,C 90.000,E1 219.277} C_DIS
LIN {X 0.075,Y -469.571,Z 454.006,A 0.000,B 0.000,C 90.000,E1 217.076} C_DIS
LIN {X 0.104,Y -465.465,Z 453.996,A 0.000,B 0.000,C 90.000,E1 215.185} C_DIS
LIN {X -0.091,Y -460.175,Z 453.982,A 0.000,B 0.000,C 90.000,E1 212.673} C_DIS
LIN {X 0.000,Y -456.325,Z 453.971,A 0.000,B 0.000,C 90.000,E1 210.747} C_DIS
LIN {X -0.069,Y -454.455,Z 453.966,A 0.000,B 0.000,C 90.000,E1 209.795} C_DIS
LIN {X 0.019,Y -449.411,Z 453.951,A 0.000,B 0.000,C 90.000,E1 207.206} C_DIS
LIN {X -0.032,Y -446.148,Z 453.942,A 0.000,B 0.000,C 90.000,E1 205.591} C_DIS
LIN {X 0.198,Y -443.585,Z 453.935,A 0.000,B 0.000,C 90.000,E1 204.259} C_DIS
LIN {X 0.158,Y -439.014,Z 453.922,A 0.000,B 0.000,C 90.000,E1 201.972} C_DIS
LIN {X -0.006,Y -434.650,Z 453.909,A 0.000,B 0.000,C 90.000,E1 199.685} C_DIS
LIN {X -0.098,Y -429.938,Z 453.895,A 0.000,B 0.000,C 90.000,E1 197.040} C_DIS
LIN {X -0.043,Y -425.791,Z 453.880,A 0.000,B 0.000,C 90.000,E1 194.356} C_DIS
LIN {X -0.094,Y -422.399,Z 453.867,A 0.000,B 0.000,C 90.000,E1 192.007} C_DIS
LIN {X 0.157,Y -418.896,Z 453.852,A 0.000,B 0.000,C 90.000,E1 189.265} C_DIS
LIN {X 0.104,Y -415.806,Z 453.837,A 0.000,B 0.000,C 90.000,E1 186.549} C_DIS
LIN {X -0.126,Y -413.290,Z 453.823,A 0.000,B 0.000,C 90.000,E1 184.188} C_DIS
LIN {X -0.057,Y -411.118,Z 453.810,A 0.000,B 0.000,C 90.000,E1 181.776} C_DIS
LIN {X -0.108,Y -409.022,Z 453.793,A 0.000,B 0.000,C 90.000,E1 178.682} C_DIS
LIN {X -0.155,Y -408.096,Z 453.781,A 0.000,B 0.000,C 90.000,E1 176.617} C_DIS
LIN {X -0.217,Y -407.377,Z 453.754,A 0.000,B 0.000,C 90.000,E1 171.781} C_DIS
LIN {X -0.118,Y -407.700,Z 453.743,A 0.000,B 0.000,C 90.000,E1 169.690} C_DIS
LIN {X -0.073,Y -409.218,Z 453.722,A 0.000,B 0.000,C 90.000,E1 165.880} C_DIS
LIN {X 0.175,Y -410.883,Z 453.706,A 0.000,B 0.000,C 90.000,E1 163.087} C_DIS
LIN {X 0.076,Y -413.555,Z 453.689,A 0.000,B 0.000,C 90.000,E1 160.007} C_DIS
LIN {X -0.089,Y -415.678,Z 453.678,A 0.000,B 0.000,C 90.000,E1 157.975} C_DIS
LIN {X -0.275,Y -418.559,Z 453.664,A 0.000,B 0.000,C 90.000,E1 155.613} C_DIS
LIN {X -0.079,Y -422.189,Z 453.649,A 0.000,B 0.000,C 90.000,E1 152.871} C_DIS
LIN {X 0.257,Y -426.099,Z 453.634,A 0.000,B 0.000,C 90.000,E1 150.127} C_DIS
LIN {X 0.199,Y -429.070,Z 453.623,A 0.000,B 0.000,C 90.000,E1 148.122} C_DIS
LIN {X 0.078,Y -432.315,Z 453.612,A 0.000,B 0.000,C 90.000,E1 146.135} C_DIS
LIN {X 0.023,Y -435.701,Z 453.601,A 0.000,B 0.000,C 90.000,E1 144.149} C_DIS
LIN {X 0.133,Y -439.839,Z 453.588,A 0.000,B 0.000,C 90.000,E1 141.823} C_DIS
LIN {X -0.225,Y -441.669,Z 453.583,A 0.000,B 0.000,C 90.000,E1 140.884} C_DIS
LIN {X -0.009,Y -444.775,Z 453.573,A 0.000,B 0.000,C 90.000,E1 139.218} C_DIS
LIN {X 0.264,Y -448.495,Z 453.563,A 0.000,B 0.000,C 90.000,E1 137.229} C_DIS
LIN {X -0.051,Y -450.770,Z 453.555,A 0.000,B 0.000,C 90.000,E1 135.972} C_DIS
LIN {X -0.029,Y -452.313,Z 453.550,A 0.000,B 0.000,C 90.000,E1 135.000} C_DIS
LIN {X 0.042,Y -454.415,Z 453.541,A 0.000,B 0.000,C 90.000,E1 133.380} C_DIS
LIN {X -0.210,Y -455.371,Z 453.536,A 0.000,B 0.000,C 90.000,E1 132.447} C_DIS
LIN {X 0.170,Y -455.879,Z 453.532,A 0.000,B 0.000,C 90.000,E1 131.757} C_DIS
LIN {X -0.067,Y -456.420,Z 453.527,A 0.000,B 0.000,C 90.000,E1 130.825} C_DIS
LIN {X 0.044,Y -456.520,Z 453.521,A 0.000,B 0.000,C 90.000,E1 129.850} C_DIS
LIN {X -0.132,Y -456.156,Z 453.516,A 0.000,B 0.000,C 90.000,E1 128.910} C_DIS
LIN {X -0.025,Y -455.400,Z 453.511,A 0.000,B 0.000,C 90.000,E1 127.935} C_DIS
LIN {X -0.124,Y -453.881,Z 453.504,A 0.000,B 0.000,C 90.000,E1 126.664} C_DIS
LIN {X 0.041,Y -452.340,Z 453.498,A 0.000,B 0.000,C 90.000,E1 125.678} C_DIS
LIN {X 0.105,Y -451.132,Z 453.495,A 0.000,B 0.000,C 90.000,E1 125.025} C_DIS
LIN {X -0.100,Y -449.837,Z 453.491,A 0.000,B 0.000,C 90.000,E1 124.405} C_DIS
LIN {X 0.011,Y -447.485,Z 453.486,A 0.000,B 0.000,C 90.000,E1 123.420} C_DIS
LIN {X -0.091,Y -444.076,Z 453.479,A 0.000,B 0.000,C 90.000,E1 122.133} C_DIS
LIN {X 0.133,Y -440.488,Z 453.471,A 0.000,B 0.000,C 90.000,E1 120.797} C_DIS
LIN {X 0.081,Y -436.601,Z 453.464,A 0.000,B 0.000,C 90.000,E1 119.489} C_DIS
LIN {X 0.024,Y -434.328,Z 453.460,A 0.000,B 0.000,C 90.000,E1 118.743} C_DIS
LIN {X -0.015,Y -434.341,Z 453.460,A 0.000,B 0.000,C 90.000,E1 118.743} C_DIS
LIN {X -0.113,Y -444.891,Z 453.438,A 0.000,B 0.000,C 90.000,E1 114.899} C_DIS
LIN {X 0.146,Y -454.003,Z 453.417,A 0.000,B 0.000,C 90.000,E1 110.972} C_DIS
LIN {X 0.257,Y -456.652,Z 453.411,A 0.000,B 0.000,C 90.000,E1 109.993} C_DIS
LIN {X 0.005,Y -457.461,Z 453.410,A 0.000,B 0.000,C 90.000,E1 109.704} C_DIS
LIN {X 0.106,Y -466.123,Z 453.387,A 0.000,B 0.000,C 90.000,E1 105.552} C_DIS
LIN {X -0.171,Y -467.693,Z 453.383,A 0.000,B 0.000,C 90.000,E1 104.954} C_DIS
LIN {X -0.214,Y -475.904,Z 453.357,A 0.000,B 0.000,C 90.000,E1 100.254} C_DIS
LIN {X 0.093,Y -476.350,Z 453.355,A 0.000,B 0.000,C 90.000,E1 99.905} C_DIS
LIN {X 0.189,Y -482.025,Z 453.330,A 0.000,B 0.000,C 90.000,E1 95.454} C_DIS
LIN {X 0.175,Y -569.440,Z 453.330,A 0.000,B 0.000,C 90.000,E1 95.454} C_DIS
LIN {X -0.232,Y -573.665,Z 453.330,A 0.000,B 0.000,C 90.000,E1 95.448} C_DIS
LIN {X -0.060,Y -578.400,Z 453.330,A 0.000,B 0.000,C 90.000,E1 95.334} C_DIS
LIN {X -0.123,Y -581.081,Z 453.329,A 0.000,B 0.000,C 90.000,E1 95.277} C_DIS
LIN {X 0.225,Y -586.950,Z 453.328,A 0.000,B 0.000,C 90.000,E1 95.049} C_DIS
LIN {X -0.035,Y -593.184,Z 453.327,A 0.000,B 0.000,C 90.000,E1 94.821} C_DIS
LIN {X -0.129,Y -599.328,Z 453.325,A 0.000,B 0.000,C 90.000,E1 94.531} C_DIS
LIN {X -0.054,Y -602.311,Z 453.324,A 0.000,B 0.000,C 90.000,E1 94.359} C_DIS
LIN {X 0.090,Y -606.637,Z 453.323,A 0.000,B 0.000,C 90.000,E1 94.073} C_DIS
LIN {X -0.073,Y -612.111,Z 453.320,A 0.000,B 0.000,C 90.000,E1 93.669} C_DIS
LIN {X -0.067,Y -614.461,Z 453.319,A 0.000,B 0.000,C 90.000,E1 93.440} C_DIS
LIN {X 0.263,Y -618.071,Z 453.317,A 0.000,B 0.000,C 90.000,E1 93.037} C_DIS
LIN {X -0.021,Y -619.773,Z 453.316,A 0.000,B 0.000,C 90.000,E1 92.808} C_DIS
LIN {X 0.144,Y -621.803,Z 453.314,A 0.000,B 0.000,C 90.000,E1 92.407} C_DIS
LIN {X -0.301,Y -623.546,Z 453.311,A 0.000,B 0.000,C 90.000,E1 92.064} C_DIS
LIN {X 0.050,Y -624.573,Z 453.310,A 0.000,B 0.000,C 90.000,E1 91.776} C_DIS
LIN {X 0.097,Y -625.812,Z 453.307,A 0.000,B 0.000,C 90.000,E1 91.260} C_DIS
LIN {X 0.155,Y -626.311,Z 453.304,A 0.000,B 0.000,C 90.000,E1 90.745} C_DIS
LIN {X -0.126,Y -626.366,Z 453.303,A 0.000,B 0.000,C 90.000,E1 90.516} C_DIS
LIN {X -0.060,Y -626.104,Z 453.300,A 0.000,B 0.000,C 90.000,E1 90.000} C_DIS
LIN {X 0.005,Y -625.094,Z 453.297,A 0.000,B 0.000,C 90.000,E1 89.484} C_DIS
LIN {X 0.063,Y -623.388,Z 453.294,A 0.000,B 0.000,C 90.000,E1 88.969} C_DIS
LIN {X -0.224,Y -622.426,Z 453.293,A 0.000,B 0.000,C 90.000,E1 88.740} C_DIS
LIN {X -0.184,Y -620.038,Z 453.290,A 0.000,B 0.000,C 90.000,E1 88.224} C_DIS
LIN {X 0.160,Y -618.355,Z 453.289,A 0.000,B 0.000,C 90.000,E1 87.936} C_DIS
LIN {X 0.010,Y -617.424,Z 453.288,A 0.000,B 0.000,C 90.000,E1 87.822} C_DIS
LIN {X -0.141,Y -616.697,Z 453.287,A 0.000,B 0.000,C 90.000,E1 87.707} C_DIS
LIN {X 0.027,Y -613.306,Z 453.284,A 0.000,B 0.000,C 90.000,E1 87.192} C_DIS
LIN {X -0.291,Y -611.091,Z 453.283,A 0.000,B 0.000,C 90.000,E1 86.963} C_DIS
LIN {X -0.136,Y -607.532,Z 453.281,A 0.000,B 0.000,C 90.000,E1 86.560} C_DIS
LIN {X 0.304,Y -606.188,Z 453.280,A 0.000,B 0.000,C 90.000,E1 86.388} C_DIS
LIN {X 0.174,Y -600.165,Z 453.278,A 0.000,B 0.000,C 90.000,E1 85.927} C_DIS
LIN {X -0.073,Y -594.932,Z 453.276,A 0.000,B 0.000,C 90.000,E1 85.641} C_DIS
LIN {X 0.207,Y -589.491,Z 453.274,A 0.000,B 0.000,C 90.000,E1 85.355} C_DIS
LIN {X -0.194,Y -582.976,Z 453.273,A 0.000,B 0.000,C 90.000,E1 85.122} C_DIS
LIN {X 0.228,Y -580.901,Z 453.272,A 0.000,B 0.000,C 90.000,E1 85.008} C_DIS
LIN {X 0.167,Y -576.490,Z 453.272,A 0.000,B 0.000,C 90.000,E1 84.894} C_DIS
LIN {X 0.016,Y -569.975,Z 453.271,A 0.000,B 0.000,C 90.000,E1 84.780} C_DIS
LIN {X -0.140,Y -563.466,Z 453.271,A 0.000,B 0.000,C 90.000,E1 84.723} C_DIS
LIN {X -0.168,Y -485.478,Z 453.271,A 0.000,B 0.000,C 90.000,E1 84.723} C_DIS
LIN {X 0.002,Y -484.684,Z 453.253,A 0.000,B 0.000,C 90.000,E1 81.602} C_DIS
LIN {X -0.098,Y -480.606,Z 453.228,A 0.000,B 0.000,C 90.000,E1 76.992} C_DIS
LIN {X 0.227,Y -480.242,Z 453.226,A 0.000,B 0.000,C 90.000,E1 76.645} C_DIS
LIN {X 0.116,Y -474.071,Z 453.200,A 0.000,B 0.000,C 90.000,E1 72.000} C_DIS
LIN {X 0.145,Y -465.510,Z 453.172,A 0.000,B 0.000,C 90.000,E1 66.975} C_DIS
LIN {X 0.107,Y -459.931,Z 453.158,A 0.000,B 0.000,C 90.000,E1 64.409} C_DIS
LIN {X 0.067,Y -459.957,Z 453.158,A 0.000,B 0.000,C 90.000,E1 64.409} C_DIS
LIN {X 0.242,Y -469.555,Z 453.150,A 0.000,B 0.000,C 90.000,E1 62.999} C_DIS
LIN {X 0.108,Y -475.011,Z 453.146,A 0.000,B 0.000,C 90.000,E1 62.231} C_DIS
LIN {X -0.193,Y -482.153,Z 453.140,A 0.000,B 0.000,C 90.000,E1 61.179} C_DIS
LIN {X 0.021,Y -486.768,Z 453.136,A 0.000,B 0.000,C 90.000,E1 60.383} C_DIS
LIN {X -0.172,Y -490.183,Z 453.132,A 0.000,B 0.000,C 90.000,E1 59.793} C_DIS
LIN {X 0.078,Y -493.287,Z 453.129,A 0.000,B 0.000,C 90.000,E1 59.154} C_DIS
LIN {X 0.183,Y -496.056,Z 453.125,A 0.000,B 0.000,C 90.000,E1 58.535} C_DIS
LIN {X 0.049,Y -498.488,Z 453.122,A 0.000,B 0.000,C 90.000,E1 57.946} C_DIS
LIN {X 0.194,Y -500.533,Z 453.119,A 0.000,B 0.000,C 90.000,E1 57.327} C_DIS
LIN {X 0.234,Y -503.033,Z 453.114,A 0.000,B 0.000,C 90.000,E1 56.421} C_DIS
LIN {X -0.282,Y -504.359,Z 453.110,A 0.000,B 0.000,C 90.000,E1 55.881} C_DIS
LIN {X -0.198,Y -505.808,Z 453.105,A 0.000,B 0.000,C 90.000,E1 54.975} C_DIS
LIN {X -0.100,Y -506.846,Z 453.100,A 0.000,B 0.000,C 90.000,E1 54.069} C_DIS
LIN {X 0.310,Y -507.406,Z 453.095,A 0.000,B 0.000,C 90.000,E1 53.130} C_DIS
LIN {X -0.080,Y -507.722,Z 453.089,A 0.000,B 0.000,C 90.000,E1 51.984} C_DIS
LIN {X 0.042,Y -507.783,Z 453.086,A 0.000,B 0.000,C 90.000,E1 51.376} C_DIS
LIN {X 0.071,Y -507.630,Z 453.081,A 0.000,B 0.000,C 90.000,E1 50.481} C_DIS
LIN {X -0.228,Y -507.304,Z 453.076,A 0.000,B 0.000,C 90.000,E1 49.622} C_DIS
LIN {X 0.135,Y -506.246,Z 453.066,A 0.000,B 0.000,C 90.000,E1 47.796} C_DIS
LIN {X -0.012,Y -505.393,Z 453.059,A 0.000,B 0.000,C 90.000,E1 46.620} C_DIS
LIN {X 0.049,Y -504.220,Z 453.051,A 0.000,B 0.000,C 90.000,E1 45.121} C_DIS
LIN {X -0.131,Y -503.220,Z 453.044,A 0.000,B 0.000,C 90.000,E1 43.947} C_DIS
LIN {X 0.104,Y -501.674,Z 453.034,A 0.000,B 0.000,C 90.000,E1 42.123} C_DIS
LIN {X 0.009,Y -500.094,Z 453.024,A 0.000,B 0.000,C 90.000,E1 40.334} C_DIS
LIN {X 0.016,Y -498.713,Z 453.016,A 0.000,B 0.000,C 90.000,E1 38.830} C_DIS
LIN {X -0.191,Y -497.611,Z 453.009,A 0.000,B 0.000,C 90.000,E1 37.649} C_DIS
LIN {X 0.240,Y -496.127,Z 453.001,A 0.000,B 0.000,C 90.000,E1 36.091} C_DIS
LIN {X 0.094,Y -494.820,Z 452.994,A 0.000,B 0.000,C 90.000,E1 34.898} C_DIS
LIN {X 0.037,Y -492.727,Z 452.984,A 0.000,B 0.000,C 90.000,E1 33.086} C_DIS
LIN {X -0.183,Y -490.842,Z 452.975,A 0.000,B 0.000,C 90.000,E1 31.592} C_DIS
LIN {X -0.022,Y -488.507,Z 452.965,A 0.000,B 0.000,C 90.000,E1 29.745} C_DIS
LIN {X -0.116,Y -485.423,Z 452.952,A 0.000,B 0.000,C 90.000,E1 27.308} C_DIS
LIN {X 0.102,Y -482.622,Z 452.938,A 0.000,B 0.000,C 90.000,E1 24.823} C_DIS
LIN {X -0.184,Y -479.621,Z 452.919,A 0.000,B 0.000,C 90.000,E1 21.461} C_DIS
LIN {X 0.003,Y -477.948,Z 452.905,A 0.000,B 0.000,C 90.000,E1 18.960} C_DIS
LIN {X 0.224,Y -477.185,Z 452.898,A 0.000,B 0.000,C 90.000,E1 17.692} C_DIS
LIN {X 0.127,Y -476.167,Z 452.890,A 0.000,B 0.000,C 90.000,E1 16.150} C_DIS
LIN {X 0.225,Y -474.534,Z 452.876,A 0.000,B 0.000,C 90.000,E1 13.647} C_DIS
LIN {X 0.097,Y -473.459,Z 452.864,A 0.000,B 0.000,C 90.000,E1 11.478} C_DIS
LIN {X 0.144,Y -472.706,Z 452.850,A 0.000,B 0.000,C 90.000,E1 8.973} C_DIS
LIN {X 0.131,Y -472.398,Z 452.829,A 0.000,B 0.000,C 90.000,E1 5.220} C_DIS
LIN {X -0.005,Y -473.921,Z 452.805,A 0.000,B 0.000,C 90.000,E1 0.859} C_DIS
LIN {X -0.115,Y -476.011,Z 452.789,A 0.000,B 0.000,C 90.000,E1 357.936} C_DIS
LIN {X 0.194,Y -478.598,Z 452.775,A 0.000,B 0.000,C 90.000,E1 355.412} C_DIS
LIN {X 0.226,Y -481.742,Z 452.761,A 0.000,B 0.000,C 90.000,E1 352.932} C_DIS
LIN {X -0.054,Y -485.236,Z 452.747,A 0.000,B 0.000,C 90.000,E1 350.500} C_DIS
LIN {X 0.050,Y -488.714,Z 452.735,A 0.000,B 0.000,C 90.000,E1 348.342} C_DIS
LIN {X 0.062,Y -495.407,Z 452.717,A 0.000,B 0.000,C 90.000,E1 344.991} C_DIS
LIN {X -0.148,Y -502.465,Z 452.700,A 0.000,B 0.000,C 90.000,E1 342.000} C_DIS
LIN {X 0.096,Y -507.794,Z 452.688,A 0.000,B 0.000,C 90.000,E1 339.880} C_DIS
LIN {X 0.063,Y -512.496,Z 452.678,A 0.000,B 0.000,C 90.000,E1 338.103} C_DIS
LIN {X -0.152,Y -517.202,Z 452.669,A 0.000,B 0.000,C 90.000,E1 336.357} C_DIS
LIN {X 0.278,Y -521.071,Z 452.660,A 0.000,B 0.000,C 90.000,E1 334.845} C_DIS
LIN {X 0.150,Y -526.487,Z 452.649,A 0.000,B 0.000,C 90.000,E1 332.820} C_DIS
LIN {X 0.167,Y -531.852,Z 452.638,A 0.000,B 0.000,C 90.000,E1 330.795} C_DIS
LIN {X -0.306,Y -535.763,Z 452.630,A 0.000,B 0.000,C 90.000,E1 329.410} C_DIS
LIN {X 0.020,Y -539.669,Z 452.622,A 0.000,B 0.000,C 90.000,E1 327.946} C_DIS
LIN {X 0.276,Y -544.315,Z 452.613,A 0.000,B 0.000,C 90.000,E1 326.215} C_DIS
LIN {X 0.151,Y -548.202,Z 452.605,A 0.000,B 0.000,C 90.000,E1 324.815} C_DIS
LIN {X 0.218,Y -553.773,Z 452.594,A 0.000,B 0.000,C 90.000,E1 322.844} C_DIS
LIN {X -0.038,Y -560.236,Z 452.581,A 0.000,B 0.000,C 90.000,E1 320.642} C_DIS
LIN {X 0.037,Y -565.285,Z 452.572,A 0.000,B 0.000,C 90.000,E1 318.976} C_DIS
LIN {X -0.278,Y -569.380,Z 452.565,A 0.000,B 0.000,C 90.000,E1 317.634} C_DIS
LIN {X 0.239,Y -573.401,Z 452.557,A 0.000,B 0.000,C 90.000,E1 316.215} C_DIS
LIN {X -0.140,Y -578.977,Z 452.546,A 0.000,B 0.000,C 90.000,E1 314.352} C_DIS
LIN {X 0.296,Y -583.846,Z 452.537,A 0.000,B 0.000,C 90.000,E1 312.690} C_DIS
LIN {X -0.318,Y -587.131,Z 452.531,A 0.000,B 0.000,C 90.000,E1 311.676} C_DIS
LIN {X 0.331,Y -591.931,Z 452.523,A 0.000,B 0.000,C 90.000,E1 310.011} C_DIS
LIN {X -0.329,Y -594.273,Z 452.518,A 0.000,B 0.000,C 90.000,E1 309.277} C_DIS
LIN {X -0.144,Y -598.007,Z 452.511,A 0.000,B 0.000,C 90.000,E1 307.935} C_DIS
LIN {X 0.212,Y -601.804,Z 452.503,A 0.000,B 0.000,C 90.000,E1 306.583} C_DIS
LIN {X -0.204,Y -605.346,Z 452.496,A 0.000,B 0.000,C 90.000,E1 305.311} C_DIS
LIN {X 0.007,Y -608.145,Z 452.490,A 0.000,B 0.000,C 90.000,E1 304.246} C_DIS
LIN {X -0.091,Y -610.828,Z 452.485,A 0.000,B 0.000,C 90.000,E1 303.214} C_DIS
LIN {X -0.241,Y -614.632,Z 452.476,A 0.000,B 0.000,C 90.000,E1 301.671} C_DIS
LIN {X -0.311,Y -618.204,Z 452.467,A 0.000,B 0.000,C 90.000,E1 300.129} C_DIS
LIN {X -0.083,Y -622.044,Z 452.457,A 0.000,B 0.000,C 90.000,E1 298.309} C_DIS
LIN {X 0.222,Y -624.800,Z 452.450,A 0.000,B 0.000,C 90.000,E1 297.001} C_DIS
LIN {X 0.283,Y -627.311,Z 452.443,A 0.000,B 0.000,C 90.000,E1 295.720} C_DIS
LIN {X 0.072,Y -628.822,Z 452.439,A 0.000,B 0.000,C 90.000,E1 294.975} C_DIS
LIN {X 0.167,Y -630.543,Z 452.433,A 0.000,B 0.000,C 90.000,E1 293.951} C_DIS
LIN {X 0.020,Y -632.226,Z 452.428,A 0.000,B 0.000,C 90.000,E1 292.950} C_DIS
LIN {X -0.317,Y -634.147,Z 452.421,A 0.000,B 0.000,C 90.000,E1 291.716} C_DIS
LIN {X -0.028,Y -635.961,Z 452.414,A 0.000,B 0.000,C 90.000,E1 290.429} C_DIS
LIN {X 0.287,Y -637.648,Z 452.407,A 0.000,B 0.000,C 90.000,E1 289.141} C_DIS
LIN {X -0.217,Y -638.786,Z 452.401,A 0.000,B 0.000,C 90.000,E1 288.181} C_DIS
LIN {X 0.077,Y -639.597,Z 452.397,A 0.000,B 0.000,C 90.000,E1 287.402} C_DIS
LIN {X 0.217,Y -640.615,Z 452.391,A 0.000,B 0.000,C 90.000,E1 286.386} C_DIS
LIN {X 0.057,Y -641.824,Z 452.383,A 0.000,B 0.000,C 90.000,E1 284.898} C_DIS
LIN {X 0.063,Y -642.671,Z 452.376,A 0.000,B 0.000,C 90.000,E1 283.647} C_DIS
LIN {X 0.106,Y -643.441,Z 452.366,A 0.000,B 0.000,C 90.000,E1 281.895} C_DIS
LIN {X -0.185,Y -643.834,Z 452.358,A 0.000,B 0.000,C 90.000,E1 280.423} C_DIS
LIN {X 0.343,Y -643.869,Z 452.352,A 0.000,B 0.000,C 90.000,E1 279.378} C_DIS
LIN {X 0.139,Y -643.728,Z 452.347,A 0.000,B 0.000,C 90.000,E1 278.398} C_DIS
LIN {X 0.027,Y -643.337,Z 452.341,A 0.000,B 0.000,C 90.000,E1 277.409} C_DIS
LIN {X -0.180,Y -642.721,Z 452.336,A 0.000,B 0.000,C 90.000,E1 276.429} C_DIS
LIN {X 0.241,Y -641.812,Z 452.330,A 0.000,B 0.000,C 90.000,E1 275.391} C_DIS
LIN {X -0.044,Y -640.602,Z 452.325,A 0.000,B 0.000,C 90.000,E1 274.416} C_DIS
LIN {X 0.299,Y -639.194,Z 452.319,A 0.000,B 0.000,C 90.000,E1 273.383} C_DIS
LIN {X -0.013,Y -637.525,Z 452.313,A 0.000,B 0.000,C 90.000,E1 272.407} C_DIS
LIN {X -0.224,Y -634.659,Z 452.305,A 0.000,B 0.000,C 90.000,E1 270.917} C_DIS
LIN {X 0.126,Y -631.412,Z 452.297,A 0.000,B 0.000,C 90.000,E1 269.370} C_DIS
LIN {X -0.041,Y -629.720,Z 452.292,A 0.000,B 0.000,C 90.000,E1 268.625} C_DIS
LIN {X 0.214,Y -626.087,Z 452.284,A 0.000,B 0.000,C 90.000,E1 267.078} C_DIS
LIN {X 0.102,Y -622.871,Z 452.277,A 0.000,B 0.000,C 90.000,E1 265.812} C_DIS
LIN {X 0.255,Y -618.867,Z 452.268,A 0.000,B 0.000,C 90.000,E1 264.261} C_DIS
LIN {X 0.023,Y -615.474,Z 452.261,A 0.000,B 0.000,C 90.000,E1 262.996} C_DIS
LIN {X -0.195,Y -611.958,Z 452.254,A 0.000,B 0.000,C 90.000,E1 261.724} C_DIS
LIN {X 0.225,Y -608.359,Z 452.247,A 0.000,B 0.000,C 90.000,E1 260.387} C_DIS
LIN {X -0.012,Y -604.595,Z 452.240,A 0.000,B 0.000,C 90.000,E1 259.106} C_DIS
LIN {X 0.120,Y -599.926,Z 452.231,A 0.000,B 0.000,C 90.000,E1 257.521} C_DIS
LIN {X 0.156,Y -596.733,Z 452.225,A 0.000,B 0.000,C 90.000,E1 256.464} C_DIS
LIN {X 0.141,Y -593.526,Z 452.219,A 0.000,B 0.000,C 90.000,E1 255.408} C_DIS
LIN {X 0.333,Y -588.491,Z 452.210,A 0.000,B 0.000,C 90.000,E1 253.795} C_DIS
LIN {X -0.132,Y -583.351,Z 452.201,A 0.000,B 0.000,C 90.000,E1 252.236} C_DIS
LIN {X 0.191,Y -578.931,Z 452.194,A 0.000,B 0.000,C 90.000,E1 250.859} C_DIS
LIN {X 0.070,Y -574.423,Z 452.186,A 0.000,B 0.000,C 90.000,E1 249.518} C_DIS
LIN {X 0.079,Y -569.774,Z 452.179,A 0.000,B 0.000,C 90.000,E1 248.156} C_DIS
LIN {X 0.197,Y -565.874,Z 452.173,A 0.000,B 0.000,C 90.000,E1 247.050} C_DIS
LIN {X 0.278,Y -560.778,Z 452.165,A 0.000,B 0.000,C 90.000,E1 245.665} C_DIS
LIN {X -0.022,Y -556.630,Z 452.159,A 0.000,B 0.000,C 90.000,E1 244.588} C_DIS
LIN {X -0.107,Y -551.386,Z 452.151,A 0.000,B 0.000,C 90.000,E1 243.204} C_DIS
LIN {X -0.286,Y -543.943,Z 452.140,A 0.000,B 0.000,C 90.000,E1 241.257} C_DIS
LIN {X -0.108,Y -537.749,Z 452.131,A 0.000,B 0.000,C 90.000,E1 239.537} C_DIS
LIN {X 0.209,Y -531.633,Z 452.121,A 0.000,B 0.000,C 90.000,E1 237.788} C_DIS
LIN {X -0.091,Y -524.451,Z 452.110,A 0.000,B 0.000,C 90.000,E1 235.801} C_DIS
LIN {X 0.132,Y -519.303,Z 452.102,A 0.000,B 0.000,C 90.000,E1 234.322} C_DIS
LIN {X 0.111,Y -512.072,Z 452.091,A 0.000,B 0.000,C 90.000,E1 232.271} C_DIS
LIN {X -0.084,Y -503.754,Z 452.076,A 0.000,B 0.000,C 90.000,E1 229.622} C_DIS
LIN {X 0.172,Y -498.409,Z 452.066,A 0.000,B 0.000,C 90.000,E1 227.796} C_DIS
LIN {X -0.065,Y -491.496,Z 452.052,A 0.000,B 0.000,C 90.000,E1 225.405} C_DIS
LIN {X 0.049,Y -485.709,Z 452.040,A 0.000,B 0.000,C 90.000,E1 223.257} C_DIS
LIN {X -0.129,Y -480.842,Z 452.030,A 0.000,B 0.000,C 90.000,E1 221.434} C_DIS
LIN {X -0.223,Y -475.515,Z 452.018,A 0.000,B 0.000,C 90.000,E1 219.277} C_DIS
LIN {X -0.086,Y -470.367,Z 452.006,A 0.000,B 0.000,C 90.000,E1 217.076} C_DIS
LIN {X -0.008,Y -465.569,Z 451.994,A 0.000,B 0.000,C 90.000,E1 214.865} C_DIS
LIN {X 0.181,Y -460.932,Z 451.981,A 0.000,B 0.000,C 90.000,E1 212.625} C_DIS
LIN {X 0.016,Y -456.457,Z 451.969,A 0.000,B 0.000,C 90.000,E1 210.413} C_DIS
LIN {X -0.073,Y -453.238,Z 451.960,A 0.000,B 0.000,C 90.000,E1 208.821} C_DIS
LIN {X -0.047,Y -450.107,Z 451.951,A 0.000,B 0.000,C 90.000,E1 207.206} C_DIS
LIN {X -0.084,Y -446.819,Z 451.942,A 0.000,B 0.000,C 90.000,E1 205.591} C_DIS
LIN {X 0.157,Y -444.206,Z 451.935,A 0.000,B 0.000,C 90.000,E1 204.259} C_DIS
LIN {X 0.134,Y -439.642,Z 451.922,A 0.000,B 0.000,C 90.000,E1 201.972} C_DIS
LIN {X -0.013,Y -435.219,Z 451.909,A 0.000,B 0.000,C 90.000,E1 199.685} C_DIS
LIN {X -0.087,Y -430.512,Z 451.895,A 0.000,B 0.000,C 90.000,E1 197.040} C_DIS
LIN {X -0.210,Y -426.825,Z 451.882,A 0.000,B 0.000,C 90.000,E1 194.717} C_DIS
LIN {X -0.134,Y -423.370,Z 451.869,A 0.000,B 0.000,C 90.000,E1 192.355} C_DIS
LIN {X 0.214,Y -419.353,Z 451.852,A 0.000,B 0.000,C 90.000,E1 189.265} C_DIS
LIN {X 0.175,Y -416.244,Z 451.837,A 0.000,B 0.000,C 90.000,E1 186.549} C_DIS
LIN {X -0.043,Y -413.724,Z 451.823,A 0.000,B 0.000,C 90.000,E1 184.188} C_DIS
LIN {X 0.037,Y -411.262,Z 451.808,A 0.000,B 0.000,C 90.000,E1 181.432} C_DIS
LIN {X -0.030,Y -408.830,Z 451.785,A 0.000,B 0.000,C 90.000,E1 177.306} C_DIS
LIN {X -0.059,Y -407.857,Z 451.752,A 0.000,B 0.000,C 90.000,E1 171.432} C_DIS
LIN {X -0.175,Y -408.805,Z 451.731,A 0.000,B 0.000,C 90.000,E1 167.645} C_DIS
LIN {X -0.165,Y -410.018,Z 451.718,A 0.000,B 0.000,C 90.000,E1 165.227} C_DIS
LIN {X 0.231,Y -411.841,Z 451.703,A 0.000,B 0.000,C 90.000,E1 162.417} C_DIS
LIN {X 0.032,Y -414.386,Z 451.687,A 0.000,B 0.000,C 90.000,E1 159.699} C_DIS
LIN {X 0.108,Y -417.798,Z 451.670,A 0.000,B 0.000,C 90.000,E1 156.613} C_DIS
LIN {X -0.100,Y -419.532,Z 451.663,A 0.000,B 0.000,C 90.000,E1 155.281} C_DIS
LIN {X 0.172,Y -422.752,Z 451.649,A 0.000,B 0.000,C 90.000,E1 152.871} C_DIS
LIN {X -0.016,Y -425.708,Z 451.638,A 0.000,B 0.000,C 90.000,E1 150.873} C_DIS
LIN {X -0.077,Y -427.773,Z 451.631,A 0.000,B 0.000,C 90.000,E1 149.537} C_DIS
LIN {X -0.212,Y -433.103,Z 451.612,A 0.000,B 0.000,C 90.000,E1 146.215} C_DIS
LIN {X 0.000,Y -436.536,Z 451.601,A 0.000,B 0.000,C 90.000,E1 144.196} C_DIS
LIN {X -0.127,Y -440.797,Z 451.588,A 0.000,B 0.000,C 90.000,E1 141.904} C_DIS
LIN {X -0.210,Y -443.933,Z 451.579,A 0.000,B 0.000,C 90.000,E1 140.275} C_DIS
LIN {X 0.073,Y -446.495,Z 451.572,A 0.000,B 0.000,C 90.000,E1 138.933} C_DIS
LIN {X 0.054,Y -449.709,Z 451.563,A 0.000,B 0.000,C 90.000,E1 137.310} C_DIS
LIN {X -0.235,Y -452.622,Z 451.554,A 0.000,B 0.000,C 90.000,E1 135.729} C_DIS
LIN {X -0.192,Y -454.187,Z 451.549,A 0.000,B 0.000,C 90.000,E1 134.757} C_DIS
LIN {X -0.109,Y -455.932,Z 451.541,A 0.000,B 0.000,C 90.000,E1 133.461} C_DIS
LIN {X -0.061,Y -456.659,Z 451.538,A 0.000,B 0.000,C 90.000,E1 132.813} C_DIS
LIN {X 0.050,Y -457.532,Z 451.533,A 0.000,B 0.000,C 90.000,E1 131.838} C_DIS
LIN {X -0.169,Y -458.124,Z 451.527,A 0.000,B 0.000,C 90.000,E1 130.906} C_DIS
LIN {X -0.064,Y -458.262,Z 451.524,A 0.000,B 0.000,C 90.000,E1 130.253} C_DIS
LIN {X -0.304,Y -458.295,Z 451.520,A 0.000,B 0.000,C 90.000,E1 129.644} C_DIS
LIN {X -0.171,Y -457.871,Z 451.515,A 0.000,B 0.000,C 90.000,E1 128.669} C_DIS
LIN {X 0.034,Y -457.047,Z 451.509,A 0.000,B 0.000,C 90.000,E1 127.684} C_DIS
LIN {X -0.128,Y -455.904,Z 451.504,A 0.000,B 0.000,C 90.000,E1 126.744} C_DIS
LIN {X 0.063,Y -454.402,Z 451.499,A 0.000,B 0.000,C 90.000,E1 125.758} C_DIS
LIN {X 0.145,Y -453.254,Z 451.495,A 0.000,B 0.000,C 90.000,E1 125.105} C_DIS
LIN {X 0.298,Y -451.180,Z 451.490,A 0.000,B 0.000,C 90.000,E1 124.119} C_DIS
LIN {X 0.174,Y -448.711,Z 451.484,A 0.000,B 0.000,C 90.000,E1 123.166} C_DIS
LIN {X 0.095,Y -445.225,Z 451.477,A 0.000,B 0.000,C 90.000,E1 121.878} C_DIS
LIN {X -0.096,Y -442.469,Z 451.472,A 0.000,B 0.000,C 90.000,E1 120.924} C_DIS
LIN {X -0.077,Y -437.518,Z 451.463,A 0.000,B 0.000,C 90.000,E1 119.283} C_DIS
LIN {X -0.137,Y -435.026,Z 451.458,A 0.000,B 0.000,C 90.000,E1 118.487} C_DIS
LIN {X -0.177,Y -435.019,Z 451.458,A 0.000,B 0.000,C 90.000,E1 118.487} C_DIS
LIN {X 0.109,Y -444.608,Z 451.439,A 0.000,B 0.000,C 90.000,E1 114.975} C_DIS
LIN {X 0.166,Y -455.467,Z 451.414,A 0.000,B 0.000,C 90.000,E1 110.429} C_DIS
LIN {X -0.036,Y -457.256,Z 451.410,A 0.000,B 0.000,C 90.000,E1 109.812} C_DIS
LIN {X 0.032,Y -465.877,Z 451.387,A 0.000,B 0.000,C 90.000,E1 105.662} C_DIS
LIN {X 0.204,Y -467.438,Z 451.384,A 0.000,B 0.000,C 90.000,E1 105.009} C_DIS
LIN {X 0.009,Y -468.056,Z 451.382,A 0.000,B 0.000,C 90.000,E1 104.717} C_DIS
LIN {X 0.149,Y -475.694,Z 451.357,A 0.000,B 0.000,C 90.000,E1 100.310} C_DIS
LIN {X -0.014,Y -476.258,Z 451.356,A 0.000,B 0.000,C 90.000,E1 100.018} C_DIS
LIN {X 0.250,Y -482.146,Z 451.330,A 0.000,B 0.000,C 90.000,E1 95.334} C_DIS
LIN {X -0.051,Y -482.390,Z 451.327,A 0.000,B 0.000,C 90.000,E1 94.821} C_DIS
LIN {X -0.108,Y -572.300,Z 451.327,A 0.000,B 0.000,C 90.000,E1 94.821} C_DIS
LIN {X 0.174,Y -575.726,Z 451.327,A 0.000,B 0.000,C 90.000,E1 94.759} C_DIS
LIN {X -0.209,Y -580.712,Z 451.326,A 0.000,B 0.000,C 90.000,E1 94.702} C_DIS
LIN {X -0.210,Y -586.417,Z 451.325,A 0.000,B 0.000,C 90.000,E1 94.531} C_DIS
LIN {X -0.277,Y -592.569,Z 451.324,A 0.000,B 0.000,C 90.000,E1 94.302} C_DIS
LIN {X 0.085,Y -595.493,Z 451.323,A 0.000,B 0.000,C 90.000,E1 94.131} C_DIS
LIN {X 0.297,Y -601.425,Z 451.321,A 0.000,B 0.000,C 90.000,E1 93.784} C_DIS
LIN {X -0.149,Y -606.848,Z 451.319,A 0.000,B 0.000,C 90.000,E1 93.440} C_DIS
LIN {X -0.014,Y -610.657,Z 451.317,A 0.000,B 0.000,C 90.000,E1 93.094} C_DIS
LIN {X -0.206,Y -612.871,Z 451.316,A 0.000,B 0.000,C 90.000,E1 92.865} C_DIS
LIN {X -0.081,Y -615.668,Z 451.314,A 0.000,B 0.000,C 90.000,E1 92.465} C_DIS
LIN {X -0.091,Y -618.364,Z 451.311,A 0.000,B 0.000,C 90.000,E1 91.949} C_DIS
LIN {X 0.240,Y -619.292,Z 451.309,A 0.000,B 0.000,C 90.000,E1 91.661} C_DIS
LIN {X 0.252,Y -620.508,Z 451.307,A 0.000,B 0.000,C 90.000,E1 91.146} C_DIS
LIN {X 0.275,Y -621.145,Z 451.304,A 0.000,B 0.000,C 90.000,E1 90.630} C_DIS
LIN {X 0.304,Y -620.886,Z 451.301,A 0.000,B 0.000,C 90.000,E1 90.115} C_DIS
LIN {X -0.287,Y -620.014,Z 451.298,A 0.000,B 0.000,C 90.000,E1 89.656} C_DIS
LIN {X 0.037,Y -619.455,Z 451.297,A 0.000,B 0.000,C 90.000,E1 89.370} C_DIS
LIN {X -0.262,Y -618.648,Z 451.295,A 0.000,B 0.000,C 90.000,E1 89.141} C_DIS
LIN {X 0.056,Y -617.667,Z 451.294,A 0.000,B 0.000,C 90.000,E1 88.854} C_DIS
LIN {X 0.214,Y -615.493,Z 451.292,A 0.000,B 0.000,C 90.000,E1 88.453} C_DIS
LIN {X -0.096,Y -614.317,Z 451.290,A 0.000,B 0.000,C 90.000,E1 88.224} C_DIS
LIN {X 0.232,Y -612.699,Z 451.289,A 0.000,B 0.000,C 90.000,E1 87.936} C_DIS
LIN {X -0.236,Y -609.966,Z 451.287,A 0.000,B 0.000,C 90.000,E1 87.593} C_DIS
LIN {X -0.119,Y -606.733,Z 451.284,A 0.000,B 0.000,C 90.000,E1 87.192} C_DIS
LIN {X 0.136,Y -602.606,Z 451.282,A 0.000,B 0.000,C 90.000,E1 86.788} C_DIS
LIN {X 0.074,Y -599.797,Z 451.281,A 0.000,B 0.000,C 90.000,E1 86.560} C_DIS
LIN {X 0.225,Y -594.659,Z 451.279,A 0.000,B 0.000,C 90.000,E1 86.216} C_DIS
LIN {X -0.244,Y -592.531,Z 451.279,A 0.000,B 0.000,C 90.000,E1 86.159} C_DIS
LIN {X -0.213,Y -587.376,Z 451.277,A 0.000,B 0.000,C 90.000,E1 85.927} C_DIS
LIN {X 0.063,Y -582.116,Z 451.276,A 0.000,B 0.000,C 90.000,E1 85.698} C_DIS
LIN {X -0.028,Y -575.849,Z 451.275,A 0.000,B 0.000,C 90.000,E1 85.527} C_DIS
LIN {X -0.117,Y -569.318,Z 451.275,A 0.000,B 0.000,C 90.000,E1 85.412} C_DIS
LIN {X 0.098,Y -562.654,Z 451.274,A 0.000,B 0.000,C 90.000,E1 85.355} C_DIS
LIN {X 0.037,Y -485.832,Z 451.274,A 0.000,B 0.000,C 90.000,E1 85.355} C_DIS
LIN {X -0.071,Y -484.690,Z 451.254,A 0.000,B 0.000,C 90.000,E1 81.659} C_DIS
LIN {X 0.075,Y -484.058,Z 451.250,A 0.000,B 0.000,C 90.000,E1 81.027} C_DIS
LIN {X -0.161,Y -480.632,Z 451.228,A 0.000,B 0.000,C 90.000,E1 77.048} C_DIS
LIN {X 0.165,Y -480.324,Z 451.226,A 0.000,B 0.000,C 90.000,E1 76.700} C_DIS
LIN {X 0.069,Y -474.138,Z 451.200,A 0.000,B 0.000,C 90.000,E1 72.054} C_DIS
LIN {X -0.064,Y -465.610,Z 451.173,A 0.000,B 0.000,C 90.000,E1 67.050} C_DIS
LIN {X -0.153,Y -460.375,Z 451.159,A 0.000,B 0.000,C 90.000,E1 64.665} C_DIS
LIN {X -0.193,Y -460.378,Z 451.159,A 0.000,B 0.000,C 90.000,E1 64.665} C_DIS
LIN {X -0.138,Y -470.147,Z 451.151,A 0.000,B 0.000,C 90.000,E1 63.256} C_DIS
LIN {X -0.268,Y -475.710,Z 451.147,A 0.000,B 0.000,C 90.000,E1 62.487} C_DIS
LIN {X 0.286,Y -483.898,Z 451.140,A 0.000,B 0.000,C 90.000,E1 61.179} C_DIS
LIN {X 0.073,Y -487.617,Z 451.137,A 0.000,B 0.000,C 90.000,E1 60.589} C_DIS
LIN {X -0.116,Y -491.071,Z 451.133,A 0.000,B 0.000,C 90.000,E1 59.999} C_DIS
LIN {X -0.283,Y -494.267,Z 451.130,A 0.000,B 0.000,C 90.000,E1 59.410} C_DIS
LIN {X -0.172,Y -497.133,Z 451.127,A 0.000,B 0.000,C 90.000,E1 58.791} C_DIS
LIN {X 0.190,Y -500.141,Z 451.122,A 0.000,B 0.000,C 90.000,E1 57.995} C_DIS
LIN {X 0.078,Y -502.187,Z 451.119,A 0.000,B 0.000,C 90.000,E1 57.406} C_DIS
LIN {X 0.133,Y -504.640,Z 451.114,A 0.000,B 0.000,C 90.000,E1 56.501} C_DIS
LIN {X -0.091,Y -505.984,Z 451.111,A 0.000,B 0.000,C 90.000,E1 55.928} C_DIS
LIN {X 0.016,Y -507.424,Z 451.106,A 0.000,B 0.000,C 90.000,E1 55.022} C_DIS
LIN {X 0.139,Y -508.395,Z 451.101,A 0.000,B 0.000,C 90.000,E1 54.116} C_DIS
LIN {X -0.141,Y -508.922,Z 451.096,A 0.000,B 0.000,C 90.000,E1 53.256} C_DIS
LIN {X -0.010,Y -509.163,Z 451.091,A 0.000,B 0.000,C 90.000,E1 52.351} C_DIS
LIN {X 0.028,Y -509.236,Z 451.086,A 0.000,B 0.000,C 90.000,E1 51.457} C_DIS
LIN {X 0.074,Y -509.032,Z 451.081,A 0.000,B 0.000,C 90.000,E1 50.561} C_DIS
LIN {X 0.118,Y -508.675,Z 451.076,A 0.000,B 0.000,C 90.000,E1 49.666} C_DIS
LIN {X 0.287,Y -507.762,Z 451.068,A 0.000,B 0.000,C 90.000,E1 48.162} C_DIS
LIN {X 0.166,Y -506.898,Z 451.061,A 0.000,B 0.000,C 90.000,E1 46.986} C_DIS
LIN {X 0.033,Y -505.909,Z 451.055,A 0.000,B 0.000,C 90.000,E1 45.810} C_DIS
LIN {X -0.027,Y -504.354,Z 451.045,A 0.000,B 0.000,C 90.000,E1 44.028} C_DIS
LIN {X 0.111,Y -502.530,Z 451.033,A 0.000,B 0.000,C 90.000,E1 41.919} C_DIS
LIN {X -0.216,Y -501.168,Z 451.025,A 0.000,B 0.000,C 90.000,E1 40.458} C_DIS
LIN {X 0.194,Y -499.764,Z 451.016,A 0.000,B 0.000,C 90.000,E1 38.910} C_DIS
LIN {X -0.124,Y -498.371,Z 451.008,A 0.000,B 0.000,C 90.000,E1 37.443} C_DIS
LIN {X -0.078,Y -496.853,Z 451.000,A 0.000,B 0.000,C 90.000,E1 35.931} C_DIS
LIN {X 0.190,Y -495.489,Z 450.993,A 0.000,B 0.000,C 90.000,E1 34.692} C_DIS
LIN {X 0.032,Y -494.076,Z 450.986,A 0.000,B 0.000,C 90.000,E1 33.499} C_DIS
LIN {X -0.006,Y -492.625,Z 450.979,A 0.000,B 0.000,C 90.000,E1 32.291} C_DIS
LIN {X 0.029,Y -490.303,Z 450.969,A 0.000,B 0.000,C 90.000,E1 30.463} C_DIS
LIN {X -0.070,Y -488.717,Z 450.963,A 0.000,B 0.000,C 90.000,E1 29.255} C_DIS
LIN {X -0.195,Y -486.030,Z 450.951,A 0.000,B 0.000,C 90.000,E1 27.129} C_DIS
LIN {X 0.050,Y -483.264,Z 450.937,A 0.000,B 0.000,C 90.000,E1 24.643} C_DIS
LIN {X -0.196,Y -480.527,Z 450.920,A 0.000,B 0.000,C 90.000,E1 21.589} C_DIS
LIN {X 0.024,Y -478.846,Z 450.906,A 0.000,B 0.000,C 90.000,E1 19.087} C_DIS
LIN {X -0.193,Y -478.078,Z 450.899,A 0.000,B 0.000,C 90.000,E1 17.873} C_DIS
LIN {X 0.157,Y -476.844,Z 450.889,A 0.000,B 0.000,C 90.000,E1 15.969} C_DIS
LIN {X -0.142,Y -475.387,Z 450.877,A 0.000,B 0.000,C 90.000,E1 13.828} C_DIS
LIN {X 0.154,Y -474.168,Z 450.863,A 0.000,B 0.000,C 90.000,E1 11.299} C_DIS
LIN {X 0.140,Y -473.386,Z 450.849,A 0.000,B 0.000,C 90.000,E1 8.803} C_DIS
LIN {X -0.014,Y -473.202,Z 450.826,A 0.000,B 0.000,C 90.000,E1 4.759} C_DIS
LIN {X -0.130,Y -474.878,Z 450.802,A 0.000,B 0.000,C 90.000,E1 0.401} C_DIS
LIN {X -0.146,Y -478.233,Z 450.780,A 0.000,B 0.000,C 90.000,E1 356.388} C_DIS
LIN {X 0.099,Y -481.570,Z 450.764,A 0.000,B 0.000,C 90.000,E1 353.571} C_DIS
LIN {X -0.063,Y -484.595,Z 450.752,A 0.000,B 0.000,C 90.000,E1 351.432} C_DIS
LIN {X -0.194,Y -488.404,Z 450.739,A 0.000,B 0.000,C 90.000,E1 348.993} C_DIS
LIN {X -0.189,Y -495.482,Z 450.718,A 0.000,B 0.000,C 90.000,E1 345.338} C_DIS
LIN {X 0.054,Y -500.277,Z 450.707,A 0.000,B 0.000,C 90.000,E1 343.196} C_DIS
LIN {X 0.172,Y -506.228,Z 450.693,A 0.000,B 0.000,C 90.000,E1 340.786} C_DIS
LIN {X -0.070,Y -510.913,Z 450.684,A 0.000,B 0.000,C 90.000,E1 339.028} C_DIS
LIN {X 0.029,Y -514.880,Z 450.675,A 0.000,B 0.000,C 90.000,E1 337.539} C_DIS
LIN {X 0.205,Y -518.771,Z 450.667,A 0.000,B 0.000,C 90.000,E1 336.049} C_DIS
LIN {X -0.177,Y -521.930,Z 450.661,A 0.000,B 0.000,C 90.000,E1 334.921} C_DIS
LIN {X 0.255,Y -526.577,Z 450.651,A 0.000,B 0.000,C 90.000,E1 333.127} C_DIS
LIN {X -0.094,Y -530.423,Z 450.643,A 0.000,B 0.000,C 90.000,E1 331.719} C_DIS
LIN {X -0.156,Y -535.166,Z 450.633,A 0.000,B 0.000,C 90.000,E1 329.999} C_DIS
LIN {X -0.116,Y -539.896,Z 450.624,A 0.000,B 0.000,C 90.000,E1 328.280} C_DIS
LIN {X 0.119,Y -543.801,Z 450.616,A 0.000,B 0.000,C 90.000,E1 326.834} C_DIS
LIN {X -0.286,Y -548.509,Z 450.606,A 0.000,B 0.000,C 90.000,E1 325.182} C_DIS
LIN {X -0.084,Y -555.660,Z 450.592,A 0.000,B 0.000,C 90.000,E1 322.637} C_DIS
LIN {X -0.296,Y -562.188,Z 450.580,A 0.000,B 0.000,C 90.000,E1 320.436} C_DIS
LIN {X -0.186,Y -567.319,Z 450.571,A 0.000,B 0.000,C 90.000,E1 318.771} C_DIS
LIN {X 0.027,Y -572.204,Z 450.562,A 0.000,B 0.000,C 90.000,E1 317.106} C_DIS
LIN {X -0.106,Y -577.069,Z 450.553,A 0.000,B 0.000,C 90.000,E1 315.486} C_DIS
LIN {X 0.158,Y -583.609,Z 450.541,A 0.000,B 0.000,C 90.000,E1 313.299} C_DIS
LIN {X -0.284,Y -587.754,Z 450.533,A 0.000,B 0.000,C 90.000,E1 312.000} C_DIS
LIN {X -0.065,Y -592.629,Z 450.524,A 0.000,B 0.000,C 90.000,E1 310.378} C_DIS
LIN {X -0.126,Y -595.801,Z 450.518,A 0.000,B 0.000,C 90.000,E1 309.322} C_DIS
LIN {X 0.183,Y -599.585,Z 450.511,A 0.000,B 0.000,C 90.000,E1 307.971} C_DIS
LIN {X 0.096,Y -603.397,Z 450.504,A 0.000,B 0.000,C 90.000,E1 306.664} C_DIS
LIN {X -0.024,Y -607.704,Z 450.495,A 0.000,B 0.000,C 90.000,E1 305.105} C_DIS
LIN {X 0.158,Y -611.156,Z 450.488,A 0.000,B 0.000,C 90.000,E1 303.785} C_DIS
LIN {X 0.107,Y -613.779,Z 450.482,A 0.000,B 0.000,C 90.000,E1 302.752} C_DIS
LIN {X 0.085,Y -616.344,Z 450.476,A 0.000,B 0.000,C 90.000,E1 301.720} C_DIS
LIN {X -0.268,Y -619.991,Z 450.468,A 0.000,B 0.000,C 90.000,E1 300.207} C_DIS
LIN {X 0.305,Y -623.314,Z 450.459,A 0.000,B 0.000,C 90.000,E1 298.615} C_DIS
LIN {X -0.203,Y -626.647,Z 450.451,A 0.000,B 0.000,C 90.000,E1 297.129} C_DIS
LIN {X -0.133,Y -628.708,Z 450.445,A 0.000,B 0.000,C 90.000,E1 296.104} C_DIS
LIN {X -0.039,Y -630.744,Z 450.439,A 0.000,B 0.000,C 90.000,E1 295.079} C_DIS
LIN {X -0.122,Y -633.382,Z 450.431,A 0.000,B 0.000,C 90.000,E1 293.567} C_DIS
LIN {X 0.350,Y -635.009,Z 450.425,A 0.000,B 0.000,C 90.000,E1 292.514} C_DIS
LIN {X 0.020,Y -636.576,Z 450.420,A 0.000,B 0.000,C 90.000,E1 291.535} C_DIS
LIN {X -0.245,Y -638.369,Z 450.413,A 0.000,B 0.000,C 90.000,E1 290.301} C_DIS
LIN {X 0.071,Y -639.742,Z 450.407,A 0.000,B 0.000,C 90.000,E1 289.268} C_DIS
LIN {X -0.237,Y -640.650,Z 450.403,A 0.000,B 0.000,C 90.000,E1 288.544} C_DIS
LIN {X 0.107,Y -641.781,Z 450.397,A 0.000,B 0.000,C 90.000,E1 287.511} C_DIS
LIN {X 0.113,Y -642.951,Z 450.390,A 0.000,B 0.000,C 90.000,E1 286.260} C_DIS
LIN {X -0.008,Y -644.193,Z 450.382,A 0.000,B 0.000,C 90.000,E1 284.773} C_DIS
LIN {X -0.122,Y -644.969,Z 450.375,A 0.000,B 0.000,C 90.000,E1 283.536} C_DIS
LIN {X -0.076,Y -645.427,Z 450.370,A 0.000,B 0.000,C 90.000,E1 282.535} C_DIS
LIN {X -0.177,Y -645.889,Z 450.363,A 0.000,B 0.000,C 90.000,E1 281.299} C_DIS
LIN {X -0.256,Y -646.116,Z 450.357,A 0.000,B 0.000,C 90.000,E1 280.310} C_DIS
LIN {X 0.308,Y -646.084,Z 450.352,A 0.000,B 0.000,C 90.000,E1 279.265} C_DIS
LIN {X 0.229,Y -645.818,Z 450.346,A 0.000,B 0.000,C 90.000,E1 278.276} C_DIS
LIN {X 0.054,Y -645.397,Z 450.341,A 0.000,B 0.000,C 90.000,E1 277.296} C_DIS
LIN {X -0.123,Y -644.764,Z 450.335,A 0.000,B 0.000,C 90.000,E1 276.315} C_DIS
LIN {X -0.133,Y -644.091,Z 450.331,A 0.000,B 0.000,C 90.000,E1 275.568} C_DIS
LIN {X 0.310,Y -642.879,Z 450.325,A 0.000,B 0.000,C 90.000,E1 274.531} C_DIS
LIN {X 0.042,Y -641.452,Z 450.320,A 0.000,B 0.000,C 90.000,E1 273.555} C_DIS
LIN {X -0.243,Y -639.807,Z 450.314,A 0.000,B 0.000,C 90.000,E1 272.579} C_DIS
LIN {X -0.162,Y -637.438,Z 450.307,A 0.000,B 0.000,C 90.000,E1 271.318} C_DIS
LIN {X -0.270,Y -635.898,Z 450.303,A 0.000,B 0.000,C 90.000,E1 270.573} C_DIS
LIN {X -0.267,Y -633.177,Z 450.296,A 0.000,B 0.000,C 90.000,E1 269.312} C_DIS
LIN {X 0.214,Y -631.419,Z 450.292,A 0.000,B 0.000,C 90.000,E1 268.511} C_DIS
LIN {X -0.125,Y -627.729,Z 450.283,A 0.000,B 0.000,C 90.000,E1 267.020} C_DIS
LIN {X -0.209,Y -624.440,Z 450.276,A 0.000,B 0.000,C 90.000,E1 265.755} C_DIS
LIN {X -0.023,Y -620.414,Z 450.268,A 0.000,B 0.000,C 90.000,E1 264.204} C_DIS
LIN {X -0.154,Y -616.985,Z 450.261,A 0.000,B 0.000,C 90.000,E1 262.932} C_DIS
LIN {X -0.070,Y -612.715,Z 450.252,A 0.000,B 0.000,C 90.000,E1 261.376} C_DIS
LIN {X 0.021,Y -609.771,Z 450.246,A 0.000,B 0.000,C 90.000,E1 260.330} C_DIS
LIN {X -0.194,Y -605.981,Z 450.239,A 0.000,B 0.000,C 90.000,E1 259.050} C_DIS
LIN {X -0.034,Y -601.280,Z 450.230,A 0.000,B 0.000,C 90.000,E1 257.465} C_DIS
LIN {X -0.266,Y -597.238,Z 450.223,A 0.000,B 0.000,C 90.000,E1 256.172} C_DIS
LIN {X 0.019,Y -594.809,Z 450.219,A 0.000,B 0.000,C 90.000,E1 255.353} C_DIS
LIN {X 0.235,Y -589.736,Z 450.210,A 0.000,B 0.000,C 90.000,E1 253.740} C_DIS
LIN {X -0.209,Y -584.558,Z 450.201,A 0.000,B 0.000,C 90.000,E1 252.181} C_DIS
LIN {X -0.026,Y -579.173,Z 450.192,A 0.000,B 0.000,C 90.000,E1 250.550} C_DIS
LIN {X -0.139,Y -574.636,Z 450.184,A 0.000,B 0.000,C 90.000,E1 249.209} C_DIS
LIN {X -0.123,Y -569.863,Z 450.177,A 0.000,B 0.000,C 90.000,E1 247.847} C_DIS
LIN {X -0.006,Y -565.893,Z 450.171,A 0.000,B 0.000,C 90.000,E1 246.741} C_DIS
LIN {X 0.076,Y -560.733,Z 450.163,A 0.000,B 0.000,C 90.000,E1 245.357} C_DIS
LIN {X 0.094,Y -554.442,Z 450.154,A 0.000,B 0.000,C 90.000,E1 243.691} C_DIS
LIN {X -0.016,Y -548.042,Z 450.145,A 0.000,B 0.000,C 90.000,E1 242.025} C_DIS
LIN {X -0.005,Y -540.708,Z 450.134,A 0.000,B 0.000,C 90.000,E1 240.049} C_DIS
LIN {X -0.184,Y -533.536,Z 450.123,A 0.000,B 0.000,C 90.000,E1 238.074} C_DIS
LIN {X -0.119,Y -527.314,Z 450.113,A 0.000,B 0.000,C 90.000,E1 236.342} C_DIS
LIN {X -0.140,Y -522.189,Z 450.105,A 0.000,B 0.000,C 90.000,E1 234.895} C_DIS
LIN {X 0.096,Y -518.045,Z 450.098,A 0.000,B 0.000,C 90.000,E1 233.703} C_DIS
LIN {X 0.022,Y -511.922,Z 450.089,A 0.000,B 0.000,C 90.000,E1 231.949} C_DIS
LIN {X -0.054,Y -504.592,Z 450.076,A 0.000,B 0.000,C 90.000,E1 229.585} C_DIS
LIN {X -0.103,Y -499.262,Z 450.066,A 0.000,B 0.000,C 90.000,E1 227.796} C_DIS
LIN {X -0.164,Y -494.892,Z 450.057,A 0.000,B 0.000,C 90.000,E1 226.296} C_DIS
LIN {X -0.315,Y -489.008,Z 450.045,A 0.000,B 0.000,C 90.000,E1 224.190} C_DIS
LIN {X -0.055,Y -484.120,Z 450.035,A 0.000,B 0.000,C 90.000,E1 222.324} C_DIS
LIN {X -0.107,Y -478.589,Z 450.023,A 0.000,B 0.000,C 90.000,E1 220.172} C_DIS
LIN {X -0.047,Y -474.088,Z 450.013,A 0.000,B 0.000,C 90.000,E1 218.302} C_DIS
LIN {X 0.060,Y -467.706,Z 449.997,A 0.000,B 0.000,C 90.000,E1 215.471} C_DIS
LIN {X 0.051,Y -463.674,Z 449.987,A 0.000,B 0.000,C 90.000,E1 213.579} C_DIS
LIN {X 0.199,Y -459.081,Z 449.974,A 0.000,B 0.000,C 90.000,E1 211.337} C_DIS
LIN {X 0.158,Y -455.900,Z 449.965,A 0.000,B 0.000,C 90.000,E1 209.745} C_DIS
LIN {X -0.071,Y -452.057,Z 449.955,A 0.000,B 0.000,C 90.000,E1 207.847} C_DIS
LIN {X -0.068,Y -448.830,Z 449.946,A 0.000,B 0.000,C 90.000,E1 206.232} C_DIS
LIN {X 0.125,Y -444.835,Z 449.935,A 0.000,B 0.000,C 90.000,E1 204.259} C_DIS
LIN {X 0.119,Y -440.276,Z 449.922,A 0.000,B 0.000,C 90.000,E1 201.972} C_DIS
LIN {X -0.012,Y -435.794,Z 449.909,A 0.000,B 0.000,C 90.000,E1 199.685} C_DIS
LIN {X -0.067,Y -431.095,Z 449.895,A 0.000,B 0.000,C 90.000,E1 197.040} C_DIS
LIN {X 0.147,Y -427.887,Z 449.884,A 0.000,B 0.000,C 90.000,E1 195.009} C_DIS
LIN {X -0.082,Y -423.880,Z 449.869,A 0.000,B 0.000,C 90.000,E1 192.355} C_DIS
LIN {X -0.132,Y -419.846,Z 449.852,A 0.000,B 0.000,C 90.000,E1 189.321} C_DIS
LIN {X -0.162,Y -417.053,Z 449.839,A 0.000,B 0.000,C 90.000,E1 186.947} C_DIS
LIN {X 0.046,Y -414.541,Z 449.825,A 0.000,B 0.000,C 90.000,E1 184.531} C_DIS
LIN {X 0.144,Y -411.992,Z 449.810,A 0.000,B 0.000,C 90.000,E1 181.776} C_DIS
LIN {X 0.115,Y -409.711,Z 449.791,A 0.000,B 0.000,C 90.000,E1 178.339} C_DIS
LIN {X 0.093,Y -408.686,Z 449.777,A 0.000,B 0.000,C 90.000,E1 175.927} C_DIS
LIN {X 0.121,Y -408.358,Z 449.751,A 0.000,B 0.000,C 90.000,E1 171.084} C_DIS
LIN {X 0.135,Y -409.576,Z 449.728,A 0.000,B 0.000,C 90.000,E1 166.937} C_DIS
LIN {X 0.042,Y -411.570,Z 449.708,A 0.000,B 0.000,C 90.000,E1 163.504} C_DIS
LIN {X 0.113,Y -414.522,Z 449.689,A 0.000,B 0.000,C 90.000,E1 160.061} C_DIS
LIN {X -0.022,Y -416.691,Z 449.678,A 0.000,B 0.000,C 90.000,E1 158.028} C_DIS
LIN {X -0.021,Y -420.098,Z 449.663,A 0.000,B 0.000,C 90.000,E1 155.305} C_DIS
LIN {X -0.157,Y -423.818,Z 449.648,A 0.000,B 0.000,C 90.000,E1 152.615} C_DIS
LIN {X -0.130,Y -427.354,Z 449.635,A 0.000,B 0.000,C 90.000,E1 150.255} C_DIS
LIN {X 0.211,Y -429.409,Z 449.627,A 0.000,B 0.000,C 90.000,E1 148.869} C_DIS
LIN {X 0.129,Y -434.434,Z 449.611,A 0.000,B 0.000,C 90.000,E1 145.881} C_DIS
LIN {X 0.036,Y -438.568,Z 449.598,A 0.000,B 0.000,C 90.000,E1 143.577} C_DIS
LIN {X 0.250,Y -441.729,Z 449.589,A 0.000,B 0.000,C 90.000,E1 141.904} C_DIS
LIN {X 0.188,Y -444.964,Z 449.579,A 0.000,B 0.000,C 90.000,E1 140.275} C_DIS
LIN {X -0.153,Y -448.283,Z 449.570,A 0.000,B 0.000,C 90.000,E1 138.690} C_DIS
LIN {X -0.139,Y -450.933,Z 449.563,A 0.000,B 0.000,C 90.000,E1 137.391} C_DIS
LIN {X 0.236,Y -453.927,Z 449.554,A 0.000,B 0.000,C 90.000,E1 135.729} C_DIS
LIN {X -0.027,Y -455.580,Z 449.549,A 0.000,B 0.000,C 90.000,E1 134.798} C_DIS
LIN {X -0.272,Y -457.031,Z 449.544,A 0.000,B 0.000,C 90.000,E1 133.866} C_DIS
LIN {X 0.153,Y -458.260,Z 449.538,A 0.000,B 0.000,C 90.000,E1 132.852} C_DIS
LIN {X -0.020,Y -459.438,Z 449.531,A 0.000,B 0.000,C 90.000,E1 131.595} C_DIS
LIN {X 0.129,Y -460.023,Z 449.526,A 0.000,B 0.000,C 90.000,E1 130.620} C_DIS
LIN {X 0.286,Y -460.118,Z 449.521,A 0.000,B 0.000,C 90.000,E1 129.644} C_DIS
LIN {X 0.056,Y -459.963,Z 449.517,A 0.000,B 0.000,C 90.000,E1 129.036} C_DIS
LIN {X 0.181,Y -459.568,Z 449.513,A 0.000,B 0.000,C 90.000,E1 128.382} C_DIS
LIN {X 0.044,Y -458.708,Z 449.508,A 0.000,B 0.000,C 90.000,E1 127.443} C_DIS
LIN {X -0.104,Y -457.514,Z 449.503,A 0.000,B 0.000,C 90.000,E1 126.503} C_DIS
LIN {X 0.102,Y -455.955,Z 449.497,A 0.000,B 0.000,C 90.000,E1 125.518} C_DIS
LIN {X 0.031,Y -454.004,Z 449.492,A 0.000,B 0.000,C 90.000,E1 124.565} C_DIS
LIN {X 0.103,Y -452.537,Z 449.489,A 0.000,B 0.000,C 90.000,E1 123.913} C_DIS
LIN {X 0.081,Y -449.153,Z 449.481,A 0.000,B 0.000,C 90.000,E1 122.625} C_DIS
LIN {X 0.077,Y -444.567,Z 449.472,A 0.000,B 0.000,C 90.000,E1 121.003} C_DIS
LIN {X -0.245,Y -439.515,Z 449.463,A 0.000,B 0.000,C 90.000,E1 119.411} C_DIS
LIN {X 0.004,Y -435.732,Z 449.457,A 0.000,B 0.000,C 90.000,E1 118.180} C_DIS
LIN {X 0.170,Y -435.736,Z 449.457,A 0.000,B 0.000,C 90.000,E1 118.153} C_DIS
LIN {X 0.152,Y -444.273,Z 449.439,A 0.000,B 0.000,C 90.000,E1 115.079} C_DIS
LIN {X 0.006,Y -445.125,Z 449.438,A 0.000,B 0.000,C 90.000,E1 114.771} C_DIS
LIN {X 0.113,Y -454.299,Z 449.416,A 0.000,B 0.000,C 90.000,E1 110.865} C_DIS
LIN {X -0.196,Y -456.967,Z 449.411,A 0.000,B 0.000,C 90.000,E1 109.939} C_DIS
LIN {X 0.043,Y -458.234,Z 449.407,A 0.000,B 0.000,C 90.000,E1 109.268} C_DIS
LIN {X 0.241,Y -466.389,Z 449.386,A 0.000,B 0.000,C 90.000,E1 105.426} C_DIS
LIN {X -0.035,Y -467.907,Z 449.382,A 0.000,B 0.000,C 90.000,E1 104.828} C_DIS
LIN {X -0.007,Y -475.477,Z 449.358,A 0.000,B 0.000,C 90.000,E1 100.433} C_DIS
LIN {X -0.169,Y -476.122,Z 449.356,A 0.000,B 0.000,C 90.000,E1 100.141} C_DIS
LIN {X 0.114,Y -482.038,Z 449.330,A 0.000,B 0.000,C 90.000,E1 95.454} C_DIS
LIN {X -0.063,Y -482.755,Z 449.323,A 0.000,B 0.000,C 90.000,E1 94.131} C_DIS
LIN {X -0.106,Y -574.355,Z 449.323,A 0.000,B 0.000,C 90.000,E1 94.131} C_DIS
LIN {X 0.141,Y -578.894,Z 449.323,A 0.000,B 0.000,C 90.000,E1 94.073} C_DIS
LIN {X -0.188,Y -580.867,Z 449.323,A 0.000,B 0.000,C 90.000,E1 94.073} C_DIS
